(* CODESYS project geral_v2_1_0.library
   DefaultNamespace: Teknike_Geral
   DocFormat: reStructuredText
   Description: FBs de uso geral
   Author: Tiago B, Cunico
   Title: Geral
   Version: 2.1.0
   Company: Teknike
   Placeholder: Teknike_Geral

Project tree, tasks and I/O mapping:
  libraries: OSCAT - AixOCAT, * (RWTH Aachen University - E.ON Energy Research Center); Tc2_EtherCAT, * (Beckhoff Automation GmbH); Tc2_IoFunctions, * (Beckhoff Automation GmbH); Tc2_Standard, * (Beckhoff Automation GmbH); Tc2_System, * (Beckhoff Automation GmbH); Tc2_Utilities, * (Beckhoff Automation GmbH); Tc3_Database, * (Beckhoff Automation GmbH); Tc3_IPCDiag, * (Beckhoff Automation GmbH); Tc3_Module, * (Beckhoff Automation GmbH)
  DUTs/
    Ethercat/
      Cartoes/
      EtherCAT Diag/
        data type E_EcCommState
        data type ST_EcMasterDevState
        data type ST_PortAddr
        data type ST_SlaveState
        data type ST_SlaveStateInfo
        data type ST_SlaveStateInfoScanned
        data type ST_TopologyData
    data type st_Coluna
  FBs/
    Alarmes/
      GerenciadorSQL/
        data type EventosSQL
        function block FB_GerenciadorDeAlarmesSQL [ST]: FazTimeStamp, GeraTabela, GravaHistorico, LeHistorico
      GerenciadorV2/
        Duts/
          data type ST_Alarmes_Historico_V2
          data type ST_Alarmes_Online_V2
          data type ST_Alarmes_V2
        Mensagens/
          function block FB_MensagemMudouBool [ST]
          function block FB_MensagemMudouInt [ST]
          function block FB_MensagemMudouReal [ST]
        function block FB_GerenciadorAlarmesV2 [ST]: DesceAlarme, SobeAlarme
    Controle/
      BotaoDeParada/
        function block FB_BotaoParada [ST]
        data type st_BotaoParada
      Telerruptor/
        data type ConfigTelerruptor
        data type ConfigTelerruptorDB
        data type enum_GravaNomes
        data type enum_LeituradosNomes
        function block FB_IniciaOsBlocosDeConfigDoTelerruptor [ST]: GeraOsTelerruptores, GeraTabela, GravaValores, LeNomes
        function block FB_Telerruptor [ST]
        data type stTelerruptor
      function block FB_Cascata [ST]
      function block FB_Cascata1Ligado [ST]
      function block FB_ContaRPMporPulso [ST]
      function block FB_ControleTorreLuminosa [ST]
      function block FB_ControleTorreLuminosaV2 [ST]
      function block FB_TimerOnOff [ST]
      function block FB_TriggerDuplo [ST]
    CSV/
      data type eStatusCSV
      function block FB_ControleCSV [ST]: ExecutaEstado, TrocaEstado
      function block FB_EscreveCSV [ST]
      function block FB_EscreveCSVPonteiro [ST]
      function block FB_LeCSV [ST]
      data type st_ControleCSV
    Diagnostico/
      CAN/
        Sts/
          data type st_Diag_CAN
        function block fb_Diag_CAN [ST]
      Ethercat/
        function block FB_EtherCATDiag [ST]: M_CheckMasterDevState, M_GetScannedSlaveName_8, M_GetSlaveAdresses_1, M_GetSlaveIdentity_6, M_GetSlaveName_7, M_GetSlaveStates_2, M_GetTopoData_4, M_GetTopoDataLen_3, M_ScanSlaves_5
        function block FB_EtherCATFrameDiag [ST]
        data type st_DiagnosticoEthercat
      Ethernet_PCgeral/
        function block FB_Diag_Geral [ST]
        data type st_Diag_Ethernet
        data type st_Diag_PC_Geral
      KPI/
        function block FB_KPI_Geral [ST]
        data type st_KPI_Geral
    EAP/
      function block FB_HarmonizaVariavel_Bool [ST]
      function block FB_HarmonizaVariavel_Int [ST]
      function block FB_HarmonizaVariavel_Real [ST]
      function block FB_HeartBeat [ST]
    Emergencia/
      Sts/
        data type st_Emergencia
        data type st_Emergencia_Banco
        data type st_Emergencia_Config
        data type st_Emergencia_Entrada
        data type st_Emergencia_Saida
        data type st_TC_SAFE
      function block FB_Emergencia [ST]: AjeitaEntrada, AjeitaSaida, CalculaKPIs, FirstScan, Timers
    Geral/
      function block FB_FFT [ST]
      function block FB_HorimetroTime_Otimizado [ST]
      function block FB_HorimetroTime_Preciso [ST]
      function block FB_RodaTextoString [ST]
      function block FB_SalvaPersistentesEHoraAgora [ST]
    Graficos/
      GraficoTF2000/
        function block FB_GraficoTF2000 [ST]
        data type ST_Grafico
    Totalizador/
      Vazao/
        function block FB_TotalizadorVazao [ST]
        data type st_HistoricoHidrometro
    Valvulas/
      Proporcional/
        function block fb_ValvulaProporcional [ST]
        data type st_ValvulaProporcional
      Valvula/
        STs/
          data type st_EntradaValvula
          data type st_SaidaValvula
          data type st_Valvula
        function block FB_ControleValvula [ST]: Controle, Status
  FUNs/
    TempoParaString/
      function F_TempoEmStringAteHoras [ST]
    function F_ConcatArray [ST]
    function F_ConcatArray1000 [ST]
    function F_ConcatArray10000 [ST]
    function F_EntradaEmPorcentagem [ST]
    function F_EstruturaDiferente [ST]
    function F_LimpaArrayString [ST]
    function F_LimpaDataBase [ST]
    function F_MaisOuMenos [ST]
    function F_RetiraCasa [ST]
    function F_StringSeparadorArrayInt [ST]
    function F_StringSeparadorArrayInt_1 [ST]
  POUs/
    global variables GVL_BlibliotecaGeral
    program Main [ST]
    program ValidaLicensa [ST]: Licensas, Tempos
  Project Information/
    function F_GetCompany [ST]
    function F_GetTitle [ST]
    function F_GetVersion [ST]
  Version/
    global variables Global_Version
  VISUs/
*)

// DUTs/Ethercat/EtherCAT Diag/E_EcCommState
TYPE E_EcCommState : (
	eEcState_UNDEFINED 	:= 0,
	eEcState_INIT 		:= 1,
	eEcState_PREOP 		:= 2,
	eEcState_BOOT 		:= 3,
	eEcState_SAFEOP 	:= 4,
	eEcState_OP 		:= 8
);
END_TYPE

// DUTs/Ethercat/EtherCAT Diag/ST_EcMasterDevState
TYPE ST_EcMasterDevState :
STRUCT
	eEcState	 		: E_EcCommState;
	nReserved			: ARRAY [0..2] OF UINT;

	bLinkError			: BOOL;
	bResetRequired		: BOOL;
	bMissFrmRedMode		: BOOL;
	bWatchdogTriggerd	: BOOL;
	bDriverNotFound		: BOOL;
	bResetActive		: BOOL;
	bAtLeastOneNotInOp	: BOOL;
	bDcNotInSync		: BOOL;
END_STRUCT
END_TYPE

// DUTs/Ethercat/EtherCAT Diag/ST_PortAddr
TYPE ST_PortAddr :
STRUCT
	portA : UINT;
	portB : UINT;
	portC : UINT;
	portD : UINT;
END_STRUCT
END_TYPE

// DUTs/Ethercat/EtherCAT Diag/ST_SlaveState
TYPE ST_SlaveState :
STRUCT
	(* slave state *)
	eEcState 		: E_EcCommState;
	nReserved		: UINT;
	bError			: BOOL;
	bInvalidVPRS	: BOOL;
	nReserved2		: UINT;

	(* link state *)
	bNoCommToSlave	: BOOL;
	bLinkError		: BOOL;
	bMissingLink	: BOOL;
	bUnexpectedLink	: BOOL;
	bPortA			: BOOL;
	bPortB			: BOOL;
	bPortC			: BOOL;
	bPortD			: BOOL;
END_STRUCT
END_TYPE

// DUTs/Ethercat/EtherCAT Diag/ST_SlaveStateInfo
TYPE ST_SlaveStateInfo :
STRUCT
	nIndex 			: DINT;
	sName 			: STRING; 		(* name of slave given in System Manager *)
	sType 			: STRING;		(* type of slave, e.g. EK1100*)
	nECAddr 		: UINT;			(* EtherCAT Slave Addr *)
	bDiagData		: BOOL;			(* DiagData in Slave State *)
	stPortCRCErrors	: ST_EcCrcErrorEx;(* Slave CRC-Errors, separate for each Port *)
	nSumCRCErrors	: UDINT;		(* Slave CRC-Errors, sum of all Ports *)
	stState 		: ST_SlaveState;(* EtherCAT State and Link state*)
END_STRUCT
END_TYPE

// DUTs/Ethercat/EtherCAT Diag/ST_SlaveStateInfoScanned
TYPE ST_SlaveStateInfoScanned :
STRUCT
	nIndex 			: DINT;
	sName 			: STRING; 		(* name of slave given in System Manager *)
	sType 			: STRING;		(* type of slave, e.g. EK1100*)
	nECAddr 		: UINT;			(* EtherCAT Slave Addr *)
	bDifferentName	: BOOL;			(* Name of Scanned configuration differs from Configured configuration *)
	bDifferentType	: BOOL;			(* Type Of Scanned configuration differs from Configured configuration *)
	bDifferentAddr	: BOOL;			(* EcAddress of Scanned configuration differs from Configured configuration *)
END_STRUCT
END_TYPE

// DUTs/Ethercat/EtherCAT Diag/ST_TopologyData
TYPE ST_TopologyData :
STRUCT
	iOwnPhysicalAddr 	: UINT;
	iOwnAutoIncAddr		: UINT;
	stPhysicalAddr		: ST_PortAddr;
	stAutoIncAddr		: ST_PortAddr;
	iPortDelay			: ARRAY [0..2] OF UDINT; (* EC_AD, EC_DB, EC_BC *)
	iReserved			: ARRAY [0..7] OF UDINT;
END_STRUCT
END_TYPE

// DUTs/st_Coluna
TYPE st_Coluna :
STRUCT
	
	xComeca : BOOL;
	iOrdemCorLiga : ARRAY[1..6] OF INT; // array de qual corres ligam em qual ordem, 0 -> desligado 1 -> vermelho 2 -> amarelo 3 -> verde 4 -> azul 5 -> buzzer, se quiser que mais de um acione ao mesmo tempo so colocar os dois juntos tipo, verde e amarelo é 24 ou 42
	tTempoDeCadaAcionamento : ARRAY[1..6] OF TIME; // tempo que vai ser usado para cada item do iOrdemCorLiga
	

	xVermelho : BOOL;
	xAmarelo : BOOL;
	xAzul : BOOL;
	xVerde : BOOL;
	xBuzzer : BOOL;
	xErro : BOOL;
END_STRUCT
END_TYPE

// FBs/Alarmes/GerenciadorSQL/EventosSQL
TYPE EventosSQL :
STRUCT
	
	ID 				:	T_ULARGE_INTEGER;
	Data_On			:	STRING(80);	//Data de entrada do evento
	Hora_On			:	STRING(80);	//Hora de entrada do evento
	Data_Off		:	STRING(80);	//Data de saida do evento
	Hora_Off		:	STRING(80);	//Hora de saida do evento
	Tipo			:	INT;	//Hora de saida do evento
	TAG				:	STRING(80);	// tago do que deu problema
	Texto 			:	STRING(80);	// texto do alarme
	Usuario			:	STRING(80);	//UsuárioLogado
	Grupo			:	INT;			//Byte do grupo
	TimesTamp 		:	DT;



END_STRUCT
END_TYPE

// FBs/Alarmes/GerenciadorV2/Duts/ST_Alarmes_Historico_V2
TYPE ST_Alarmes_Historico_V2 : STRUCT

		sData_on  : STRING(20);  //Data de entrada do evento
		sData_off : STRING(20);  //Data de saida do evento
		sHora_on  : STRING(20);  //Hora de entrada do evento
		sHora_off : STRING(20);  //Hora de saida do evento
		iStatus   : INT;         //Byte do grupo
		sUsuario  : STRING;      //UsuárioLogado
		sTAG      : STRING;      //tag do que foi afetado
		sTexto    : STRING(255); //texto em si
		iTipo     : INT;         //mensagem ou alarme

	END_STRUCT
END_TYPE

// FBs/Alarmes/GerenciadorV2/Duts/ST_Alarmes_Online_V2
TYPE ST_Alarmes_Online_V2 : STRUCT

		sData          : STRING(20); //Hora de entrada do alarme
		sHora          : STRING(20); //Hora de saida do alarme
		sMensagem      : STRING(255); // mensagme que aparece na tela
		sUser          : STRING; // usuario
		iStatus        : INT; // se foi reconhecido como que ta
		iIdentificador : INT; // pra controle interno
		sTAG           : STRING; // tag do que foi afetado
		iTipo          : INT; // mensagem ou alarme

	END_STRUCT
END_TYPE

// FBs/Alarmes/GerenciadorV2/Duts/ST_Alarmes_V2
TYPE ST_Alarmes_V2 : STRUCT
		xAtivo : BOOL;
		sTexto : STRING(255);
		iTipo  : INT;
		sTAG   : STRING;
	END_STRUCT
END_TYPE

// FBs/Controle/BotaoDeParada/st_BotaoParada
TYPE st_BotaoParada :
STRUCT
	xSinalBP_IN		: BOOL;
	xSinalBP_OUT	: BOOL;
	xLedBP			: BOOL;
END_STRUCT
END_TYPE

// FBs/Controle/Telerruptor/ConfigTelerruptor
TYPE ConfigTelerruptor :
STRUCT RETAIN PERSISTENT
		sNome_Funcao				: STRING;
		rTempoTelerruptorAcionado 	: REAL;
END_STRUCT
END_TYPE

// FBs/Controle/Telerruptor/ConfigTelerruptorDB
TYPE ConfigTelerruptorDB :
STRUCT
	Telerruptor: DINT;
	Tag: STRING(80);
	Funcao: STRING(80);
END_STRUCT
END_TYPE

// FBs/Controle/Telerruptor/enum_GravaNomes
{attribute 'qualified_only'}
{attribute 'strict'}
TYPE enum_GravaNomes :
(
	eEsperando := 0,
	eAbreConexao := 1,
	eGravaNomes := 2,
	eCriaComando := 3,
	eFechaConexao := 4,
	eParado := 100
);
END_TYPE

// FBs/Controle/Telerruptor/enum_LeituradosNomes
{attribute 'qualified_only'}
{attribute 'strict'}
TYPE enum_LeituradosNomes :
(
	eEsperando := 0,
	eAbreConexao := 1,
	eLeOsNomes := 2,
	eMonitoraTrocaDeNomes := 3,
	eFechaConexao := 4,
	eParado := 100
);
END_TYPE

// FBs/Controle/Telerruptor/stTelerruptor
TYPE stTelerruptor :
STRUCT
	xFeedBackTelerruptor 		: BOOL;
	xLigaIHM		 			: BOOL;
	xLigaBotoeira				: BOOL;
	xLigaInterruptor			: BOOL;
	xAcionaTelerruptor			: BOOL;
	Config						: ConfigTelerruptor;
END_STRUCT
END_TYPE

// FBs/CSV/eStatusCSV
//{attribute 'qualified_only'}
{attribute 'strict'}
TYPE eStatusCSV :
(
	Esperando := 0,
	ChecandoCaminhoGeral,
	ChecandoCaminhoEspecifico,
	Gravando,
	lendoArquivos,
	Lendo,
	Erro
);
END_TYPE

// FBs/CSV/st_ControleCSV
TYPE st_ControleCSV :
STRUCT
	
	xLeCSV 						: BOOL;
	xEscreveCSV 				: BOOL;
	xEscolhidoArquivo			: BOOL;
	
	sArquivosSelecionado		: STRING(255);

	xEscritaOcupado 			: BOOL;
	xLeituraOcupado 			: BOOL;
	
	
	iTotalLeitura 				: INT;
	iAtualLeitura 				: INT;
	iTotalEscrita 				: INT;
	iAtualEscrita 				: INT;
	sArquivos					: ARRAY[1..20]  OF STRING(255);
	
	sStado : eStatusCSV;

END_STRUCT
END_TYPE

// FBs/Diagnostico/CAN/Sts/st_Diag_CAN
TYPE st_Diag_CAN :
	STRUCT
		//Linkar no device
		usError				AT %I*	: USINT;	// numero de Box com erro
		uCanState			AT %I*	: UINT;		// gera outros bits
		usRxErrorCounter	AT %I*	: USINT;	// contagem 
		usTxErrorCounter	AT %I*	: USINT;	// contagem
		diagFlag			AT %I*	: BIT;

		//Linkar nos nos
		uNodeState AT %I* : ARRAY[1..126] OF USINT;

		//Gerado apartir do CAN state
		xBusOFF			: BOOL;
		xCanWarning		: BOOL;
		xRxOverrun		: BOOL;
		xCANSendError	: BOOL;
		xFilaRxOverflow	: BOOL;
		xFilaTxOverflow	: BOOL;

		xNoOk		: ARRAY[1..126] OF BOOL;
		sEstadoNo	: ARRAY[1..126] OF STRING;

	END_STRUCT
END_TYPE

// FBs/Diagnostico/Ethercat/st_DiagnosticoEthercat
TYPE st_DiagnosticoEthercat :
	STRUCT

		(* ******************* EtherCAT Frame ***************************** *)
		fbEtherCATFrameDiag	: FB_EtherCATFrameDiag;	// frame diagnostic 
		wFrmXWcState AT %I*	: WORD;					// link to task related ethercat frame state (Frm1WcState)
		wReqZeroMask		: WORD := 16#FFFF;		// clear bit to ignore datagram error of Frm1WcState
		bFrameWcStateOK		: BOOL;					// this frame is OK 

		(* ******************* EtherCAT Diag ***************************** *)
		bEtherCATOK				: BOOL;					// no problem on EtherCAT
		bFrameWcStateError		: BOOL;					// at least one fram with error
		bSlaveCountError		: BOOL;					// EtherCAT slave count mismatch (# of cfg slaves <> # of found slaves)
		bMasterDevStateError	: BOOL;					// EtherCAT master device state signals error
		bBarramentoInterrompido	: BOOL;					// caso o barramento esteja interrompido
		stMasterDevState		: ST_EcMasterDevState;	// device state split to a structure
		bBusy					: BOOL;					// diagnostic FB is busy
		bError					: BOOL;					// diagnostic FB has an error
		iErrorID				: UDINT;				// error ID of diagnostic FB

		(* cyclic variables from EtherCAT Master *)
		nEcMasterSlaveCount		AT %I*	: UINT;				// link to SlaveCount of EtherCAT Master (Inputs)
		nEcMasterSlaveCount2	AT %I*	: UINT;				// link to SlaveCount of EtherCAT Master (Inputs)
		nEcMasterDevState		AT %I*	: UINT;				// link to DevState of EtherCAT Master (Inputs)
		nEcMasterDeviceId		AT %I*	: UINT;				// link to DevID of EtherCAT Master (InfoData)
		arrEcMasterNetId		AT %I*	: T_AmsNetIdArr;	// link to NetID of EtherCAT Master (InfoData)
		sEcMasterNetId					: T_AmsNetId := '';
		nEcMasterSlaveCountCfg AT %I*	: UINT; // link to CfgSlaveCount of EtherCAT Master (InfoData)

		(* general variables *)
		arrDiagSlaveInfo		: ARRAY[0..255] OF ST_SlaveStateInfo;			// read in info of configured EtherCAT slaves 
		arrDiagSlaveInfoScanned	: ARRAY[0..255] OF ST_SlaveStateInfoScanned;	// read in info of scanned EtherCAT slaves

	END_STRUCT
END_TYPE

// FBs/Diagnostico/Ethernet_PCgeral/st_Diag_Ethernet
TYPE st_Diag_Ethernet :
STRUCT
	
	sNome 			: STRING;
	sNomeAdaptador 	: STRING;
	sIP				: STRING;
	sMask 			: STRING;
	xDHCP 			: BOOL;

END_STRUCT
END_TYPE

// FBs/Diagnostico/Ethernet_PCgeral/st_Diag_PC_Geral
TYPE st_Diag_PC_Geral :
STRUCT
	
	//Rede
	NumeroDePortasRede	: USINT;
	stEthernet : ARRAY[1..20] OF st_Diag_Ethernet;
	
	//CPU
	uiUsoCpu : UINT;
	iTempCpu : INT;
	rMemoriaRamUsada : REAL;
	rEspacoLivreHD : REAL;
	sNomeCPU : STRING;
	
	//Twincat
	tcVersion : STRING;
	tcAMSNetID : STRING;
	tcSystemID : STRING;
	


END_STRUCT
END_TYPE

// FBs/Diagnostico/KPI/st_KPI_Geral
TYPE st_KPI_Geral :
	STRUCT
		stGraficoIHM : ARRAY[0..2] OF ST_Grafico;
	
		rPorcEstado1	: REAL;
		rPorcEstado2	: REAL;
		rPorcEstado3	: REAL;

		tEstado1	: TIME;
		tEstado2	: TIME;
		tEstado3	: TIME;
	END_STRUCT
END_TYPE

// FBs/Emergencia/Sts/st_Emergencia
TYPE st_Emergencia :
STRUCT
	En : st_Emergencia_Entrada;
	Sa : st_Emergencia_Saida;
	Config : st_Emergencia_Config;
	Banco : st_Emergencia_Banco;
	Safe : st_TC_SAFE;
END_STRUCT
END_TYPE

// FBs/Emergencia/Sts/st_Emergencia_Banco
TYPE st_Emergencia_Banco :
STRUCT
		Emergencia	: T_ULARGE_INTEGER;
		Tag			: STRING(80);
		Funcao		: STRING(80);
		Timestamp	: DT;
END_STRUCT
END_TYPE

// FBs/Emergencia/Sts/st_Emergencia_Config
TYPE st_Emergencia_Config :
STRUCT RETAIN PERSISTENT
	xControleInterno : BOOL;
	xbypassCH2 : BOOL;
	tDiscrepancia : TIME;
	xControleTCSafe : BOOL;
END_STRUCT
END_TYPE

// FBs/Emergencia/Sts/st_Emergencia_Entrada
TYPE st_Emergencia_Entrada :
STRUCT
	xCH1 : BOOL;
	xCH2 : BOOL;
	xEmergenciaOK : BOOL; // status da emergencia, se for externa tb serve
	sNomeFuncao : STRING;
	xReset : BOOL;
	xResetFisico : BOOL;
	stHoraAgora : TIMESTRUCT;
END_STRUCT
END_TYPE

// FBs/Emergencia/Sts/st_Emergencia_Saida
TYPE st_Emergencia_Saida :
STRUCT	
	kpi : ARRAY[0..23] OF st_KPI_Geral;
	xErro : BOOL;
	xLedReset : BOOL;
	sEstadoIHM : STRING;
	iStatus : INT;//0 : desligado, 1 : OK, 2 : Esperando Reset, 3 : Desincronizado, 4 : EDM, 5 : Outro Erro
END_STRUCT
END_TYPE

// FBs/Emergencia/Sts/st_TC_SAFE
TYPE st_TC_SAFE :
STRUCT
	RESET 		AT%Q* 	: BOOL;
	EDM 		AT%Q*	: BOOL;
	RUN			AT%Q*	: BOOL;
	ERRACK		AT%Q*	: BOOL;
	
	State		AT%I*	: USINT;
	Diag		AT%I*	: UINT;
END_STRUCT
END_TYPE

// FBs/Graficos/GraficoTF2000/ST_Grafico
TYPE ST_Grafico :
STRUCT
	x : STRING;
	y : REAL;
	label : STRING(255);
	sCor : STRING(255);//Cor em Hexa
	sTipo: STRING;//sendo eles "line", "bar", "scatter", "bubble", "pie", "doughnut", "polarArea" 
END_STRUCT
END_TYPE

// FBs/Totalizador/Vazao/st_HistoricoHidrometro
TYPE st_HistoricoHidrometro :
STRUCT
	sDataHora : STRING;
	rTotal : REAL;
	rDiferenca : REAL;
END_STRUCT
END_TYPE

// FBs/Valvulas/Proporcional/st_ValvulaProporcional
TYPE st_ValvulaProporcional :
STRUCT RETAIN PERSISTENT
	xManu : BOOL;
	rValorManu : REAL;
	rValorAuto : REAL;
	
	rMinimo : REAL := 0;
	rMaximo : REAL := 32767;
	rValorDeSaida : REAL;
	
	
	rPorcentSaida : REAL;
	
	iStsValvula  : INT;
	
	sNomeFuncao : STRING;
	
	
END_STRUCT
END_TYPE

// FBs/Valvulas/Valvula/STs/st_EntradaValvula
TYPE st_EntradaValvula :
STRUCT
	xAutomaticoManual 	: BOOL;
	xLigaManu			: BOOL;
	xLigaAuto			: BOOL;
	xBloqueio			: BOOL;
	xEmergenciaOK		: BOOL;
	xFeedBackValvula	: BOOL;
	xByPassFeedBack		: BOOL;
	xResetContador		: BOOL;
	rTempoFeedBackSeg	: REAL;
	sNome_Funcao		: STRING;
	xNormalmenteAberto	: BOOL;
	i					: INT;
END_STRUCT
END_TYPE

// FBs/Valvulas/Valvula/STs/st_SaidaValvula
TYPE st_SaidaValvula :
STRUCT
	xSaidaValvula		: BOOL;
	iStsValvula			: INT;
	iSucessoAionamento	: INT;
	iFalhaAcionamento	: INT;
END_STRUCT
END_TYPE

// FBs/Valvulas/Valvula/STs/st_Valvula
TYPE st_Valvula :
STRUCT
	en : st_EntradaValvula;
	sa : st_SaidaValvula;
END_STRUCT
END_TYPE

// POUs/GVL_BlibliotecaGeral
//{attribute 'qualified_only'}
VAR_GLOBAL
	
    {attribute 'hide'} 
	{attribute 'tc_no_symbol'}
	xLicensaValida87208720 : BOOL;
	LicensaValida : BOOL;
	STCheckLicense : ST_CheckLicense;
END_VAR

// Version/Global_Version
{attribute 'TcGenerated'}
{attribute 'no-analysis'}
{attribute 'linkalways'}
// This function has been automatically generated from the project information.
VAR_GLOBAL CONSTANT
	{attribute 'const_non_replaced'}
	stLibVersion_Geral : ST_LibVersion := (iMajor := 2, iMinor := 1, iBuild := 0, iRevision := 0, nFlags := 0, sVersion := '2.1.0');
END_VAR

// FBs/Alarmes/GerenciadorSQL/FB_GerenciadorDeAlarmesSQL
//{attribute 'hide_all_locals'}
FUNCTION_BLOCK FB_GerenciadorDeAlarmesSQL
VAR_IN_OUT
	arrayAlarmes	: ARRAY[*] OF ST_Alarmes_V2;
	Alarmes_Online	: ARRAY[*] OF ST_Alarmes_Online_v2;
	HistoricoSQL	: ARRAY[*] OF EventosSQL;
	RT				: ARRAY[*] OF R_TRIG;	//
	FT				: ARRAY[*] OF F_TRIG;	//
END_VAR
VAR_INPUT
	xReconhece		: BOOL;
	sUsuario		: STRING;
	sNomeTabela		: STRING;
	iNumeroDataBase	: INT := 1;
	xCriaTabela		: BOOL;
	stTempoAgora	: TIMESTRUCT;
END_VAR
VAR_OUTPUT
	xAlarmeAtivo			: BOOL;
	xAlarmeAtivoReconhecido	: BOOL;
	sErro					: STRING;
END_VAR
VAR
	VariavelParaTamanhoNoBloco : EventosSQL;

	// Erros
	xAbaixoOk		: BOOL	:= TRUE;
	xAcimaOK		: BOOL	:= TRUE;
	xHistoricoOk	: BOOL	:= TRUE;

	// variaveis para controle dos loops
	iMaxAlarmesOnline		: INT;
	iMaxAlarmesHistorico	: INT;

	//Ler dados da tabela usando o bloco Read Struct
	fbPLCDBRead		: FB_PLCDBReadEvt(sNetID := '', tTimeout := T#30S);	//Bloco para leitura do banco de dados sem filtro
	sMensagemErro1	: STRING;											//Mensagem de erro

	ColumnNames : ARRAY[0..10] OF STRING(50) := ['ID',
												'Data_On',
												'Hora_On',
												'Data_Off',
												'Hora_Off',
												'Tipo',
												'TAG',
												'Texto',
												'Usuario',
												'Grupo',
												'Timestamp'];

	xEscreve	: BOOL;
	xAtualiza	: BOOL;

	// fb do gerenciador e auxiliares
	GerenciaAlarmes : FB_GerenciadorAlarmesV2;
	//para a data e hora
	sData	: ARRAY[1..5] OF STRING(255);
	sHora	: ARRAY[1..7] OF STRING(255);

	// para controle do historico e da escrita dele no SQL
	Alarmes_Historico		: ARRAY[0..1000] OF ST_Alarmes_Historico_v2;	// esse é o atual
	Alarmes_Historico_Bufer	: ARRAY[0..1000] OF ST_Alarmes_Historico_v2;	// Buffer pra escrita quando varios alarmes caiem de uma vez so
	Alarmes_Historico_Aux	: ARRAY[0..1000] OF ST_Alarmes_Historico_v2;	// esse é pra ver see é diferente
	tofEsperaAlarme			: TOn;

	//Gravar dados na tabela
	fbPLCDBWrite			: FB_PLCDBWriteEvt(sNetID := '', tTimeout := T#30S);	//Bloco para gravar no banco de dados
	systime					: GETSYSTEMTIME;										//Faz a leitura da data e hora do sistema
	currentTime				: T_FILETIME;
	bGravarDados			: BOOL;
	sMensagemErroEscrita	: STRING;
	AuxEscreve				: EventosSQL;
	coutBuffer				: INT;
	rtComecaEscever			: R_TRIG;
	ftTerminouDeGravar		: F_TRIG;
	xAtualizado				: BOOL;
	xTemQueEscrever			: BOOL;
	iDeslocamenteAjuste		: INT;

	// geral
	i				: INT;
	xPrimeiroScan	: BOOL := TRUE;

	rtCria			: R_TRIG;
	xCria			: BOOL;
	fbPLCDBCreate	: FB_PLCDBCreateEvt(sNetID := '', tTimeout := T#30S);

	ColumnInfo : ARRAY[0..10] OF ST_ColumnInfo := [(sName := 'ID', eType := E_ColumnType.BigInt, nLength := 8, sProperty := 'IDENTITY(1,1)'),
													(sName := 'Data_On', eType := E_ColumnType.NVarChar, nLength := 80),
													(sName := 'Hora_On', eType := E_ColumnType.NVarChar, nLength := 80),
													(sName := 'Data_Off', eType := E_ColumnType.NVarChar, nLength := 80),
													(sName := 'Hora_Off', eType := E_ColumnType.NVarChar, nLength := 80),
													(sName := 'Tipo', eType := E_ColumnType.SmallInt, nLength := 2),
													(sName := 'TAG', eType := E_ColumnType.NVarChar, nLength := 80),
													(sName := 'Texto', eType := E_ColumnType.NVarChar, nLength := 80),
													(sName := 'Usuario', eType := E_ColumnType.NVarChar, nLength := 80),
													(sName := 'Grupo', eType := E_ColumnType.SmallInt, nLength := 2),
													(
				sName := 'Timestamp',
					eType := E_ColumnType.DateTime,
					nLength := 4,
					sProperty := 'DEFAULT CURRENT_TIMESTAMP ON UPDATE CURRENT_TIMESTAMP')];
					
	tonPodeLer : TON;

END_VAR


IF xLicensaValida87208720 THEN
	

	// ve se os tamanhos dos arrays estao ok
	xAbaixoOk		:= LOWER_BOUND(arrayAlarmes, 1) = 0 AND LOWER_BOUND(arrayAlarmes, 1) = LOWER_BOUND(Alarmes_Online, 1);
	xAcimaOK		:= UPPER_BOUND(arrayAlarmes, 1) = UPPER_BOUND(Alarmes_Online, 1);
	xHistoricoOk	:= LOWER_BOUND(HistoricoSQL, 1) = 0;
	
	GeraTabela();
	
	IF xAbaixoOk AND xAcimaOK AND xHistoricoOk THEN
	
		IF xPrimeiroScan THEN
			FazTimeStamp();
			systime(timeLoDw => currentTime.dwLowDateTime, timeHiDW => currentTime.dwHighDateTime);
			// troca a variavel pra ficar bom pro sql
			AuxEscreve.Data_Off		:= '';
			AuxEscreve.Data_On		:= F_ConcatArray(sData);
			AuxEscreve.Hora_Off		:= '';
			AuxEscreve.Hora_On		:= F_ConcatArray(sHora);
			AuxEscreve.Usuario		:= '';
			AuxEscreve.Texto		:= 'CPU ligou';
			//AuxEscreve.TimesTamp	:= FILETIME_TO_DT(currentTime) - (T#3H);
	
			xAtualiza	:= TRUE;
			xEscreve	:= TRUE;
	
			iMaxAlarmesOnline		:= TO_INT(UPPER_BOUND(Alarmes_Online, 1));
			iMaxAlarmesHistorico	:= TO_INT(UPPER_BOUND(HistoricoSQL, 1));
		END_IF
	
		LeHistorico();
		FazTimeStamp();
		GravaHistorico();
	
		GerenciaAlarmes
			(
				Alarmes_Array := arrayAlarmes,
					Alarmes_Online := Alarmes_Online,
					Alarmes_Historico := Alarmes_Historico,
					RT := RT,
					FT := FT,
					xReconheceAlarmes := xReconhece,
					sData := F_ConcatArray(sData),
					sHora := F_ConcatArray(sHora),
					sUser := sUsuario,
					xAlarmeAtivo => xAlarmeAtivo,
					xAlarmeAtivoReconhecido => xAlarmeAtivoReconhecido);
	
		// independente se tem so um diferente ou varios, esse if sempre sera verdade
		IF Alarmes_Historico[0].sHora_off <> Alarmes_Historico_Aux[0].sHora_off AND NOT (Alarmes_Historico[0].sHora_off = '') THEN
			FOR i := 0 TO 1000 DO
				// quando nao tiver alguma coisa na posição do buffer ele sai do for
				IF (Alarmes_Historico_Bufer[i].sHora_off = '') THEN
					EXIT;
				END_IF
			END_FOR
			// e joga aqui o valor de i que é a primeira posição que nao tem na da no buffer
			coutBuffer := i;
			// deslocamente para ajustar o index conforme vai passando e encontrando alarmes diferentes
			iDeslocamenteAjuste := 0;
	
			// passa por todo os alarmes vendo quem ta acionado e joga no buffer
			FOR i := 0 TO 1000 DO
				IF Alarmes_Historico[i].sHora_off <> Alarmes_Historico_Aux[i - iDeslocamenteAjuste].sHora_off
						AND NOT (Alarmes_Historico[i].sHora_off = '') THEN
					Alarmes_Historico_Bufer[coutBuffer]	:= Alarmes_Historico[i];
					coutBuffer							:= coutBuffer + 1;
					iDeslocamenteAjuste					:= iDeslocamenteAjuste + 1;
				ELSE
					//IF THEN
	
					//ELSE
					EXIT;
					//END_IF
				END_IF
			END_FOR
		END_IF
	
		Alarmes_Historico_Aux := Alarmes_Historico; // atualiza para o atual
	
		// da o start quando chega o primeiro item pra ler no buffer
		rtComecaEscever(CLK := (Alarmes_Historico_Bufer[0].sHora_off <> ''), Q =>);
	
		IF rtComecaEscever.q THEN
			xEscreve	:= TRUE;
			xAtualizado	:= FALSE;
	
			// faz esse esquema a primeira vez
			// pega o tempo de agora
			systime(timeLoDw => currentTime.dwLowDateTime, timeHiDW => currentTime.dwHighDateTime);
			// troca a variavel pra ficar bom pro sql
			AuxEscreve.Data_Off	:= Alarmes_Historico_Bufer[0].sData_off;
			AuxEscreve.Data_On	:= Alarmes_Historico_Bufer[0].sData_On;
			AuxEscreve.Hora_Off	:= Alarmes_Historico_Bufer[0].sHora_Off;
			AuxEscreve.Hora_On	:= Alarmes_Historico_Bufer[0].sHora_On;
			AuxEscreve.Usuario	:= Alarmes_Historico_Bufer[0].sUsuario;
			AuxEscreve.TAG		:= Alarmes_Historico_Bufer[0].sTAG;
			AuxEscreve.Texto	:= Alarmes_Historico_Bufer[0].sTexto;
			AuxEscreve.Grupo	:= Alarmes_Historico_Bufer[0].iStatus;
			AuxEscreve.Tipo		:= Alarmes_Historico_Bufer[0].iTipo;
	
		END_IF
	
		ftTerminouDeGravar(CLK := xEscreve, Q =>);
	
		IF ftTerminouDeGravar.q THEN
			FOR i := 0 TO 999 DO
				Alarmes_Historico_Bufer[i] := Alarmes_Historico_Bufer[i + 1];
	
				IF Alarmes_Historico_Bufer[i].sHora_off = '' THEN
					EXIT;
				END_IF
			END_FOR
	
			xAtualizado := TRUE;
		END_IF
	
		IF NOT xEscreve AND xAtualizado AND Alarmes_Historico_Bufer[0].sHora_off <> '' THEN
	
			// pega o tempo de agora
			systime(timeLoDw => currentTime.dwLowDateTime, timeHiDW => currentTime.dwHighDateTime);
			// troca a variavel pra ficar bom pro sql
			AuxEscreve.Data_Off	:= Alarmes_Historico_Bufer[0].sData_off;
			AuxEscreve.Data_On	:= Alarmes_Historico_Bufer[0].sData_On;
			AuxEscreve.Hora_Off	:= Alarmes_Historico_Bufer[0].sHora_Off;
			AuxEscreve.Hora_On	:= Alarmes_Historico_Bufer[0].sHora_On;
			AuxEscreve.Usuario	:= Alarmes_Historico_Bufer[0].sUsuario;
			AuxEscreve.TAG		:= Alarmes_Historico_Bufer[0].sTAG;
			AuxEscreve.Texto	:= Alarmes_Historico_Bufer[0].sTexto;
			AuxEscreve.Grupo	:= Alarmes_Historico_Bufer[0].iStatus;
	
			//manda escrever
			xEscreve := TRUE;
			// tira esse bit pra esperar atualizar
			xAtualizado := FALSE;
		END_IF
	
		tofEsperaAlarme.in := TRUE;
	
		IF tofEsperaAlarme.q THEN
			xAtualiza			:= TRUE;
			tofEsperaAlarme.in	:= FALSE;
		END_IF
	
		tofEsperaAlarme(IN :=, PT := T#1S, Q =>, ET =>);
	
		xPrimeiroScan := FALSE;
	
	ELSE
		sErro := '';
	
		IF xHistoricoOk THEN
			sErro := 'historico precisa começar em 0';
		END_IF
	
		IF xAbaixoOk THEN
			sErro := 'tanto o online quanto o alarmes precisa começar em 0';
		END_IF
	
		IF xAcimaOK THEN
			sErro := 'tanto o online quanto o alarmes ter o mesmo tamanho';
		END_IF
	
	END_IF
	
ELSE
	ValidaLicensa();
END_IF

ACTION FazTimeStamp:



IF xPrimeiroScan THEN
	systime(timeLoDw => currentTime.dwLowDateTime, timeHiDW => currentTime.dwHighDateTime);
	AuxEscreve.TimesTamp := (FILETIME_TO_DT(currentTime));
	stTempoAgora := DT_TO_SYSTEMTIME(FILETIME_TO_DT(currentTime) - (T#3h));
END_IF

systime(timeLoDw => currentTime.dwLowDateTime, timeHiDW => currentTime.dwHighDateTime);
AuxEscreve.TimesTamp := (FILETIME_TO_DT(currentTime));


IF stTempoAgora.wDay < 10 THEN
	sData[1] := concat('0', TO_STRING(stTempoAgora.wDay));
ELSE
	sData[1] := WORD_TO_STRING(stTempoAgora.wDay);
END_IF

sData[2] := '/';

IF stTempoAgora.wMonth < 10 THEN
	sData[3] := concat('0', TO_STRING(stTempoAgora.wMonth));
ELSE
	sData[3] := WORD_TO_STRING(stTempoAgora.wMonth);
END_IF

sData[4] := '/';

sData[5] := TO_STRING(stTempoAgora.wYear);

IF stTempoAgora.wHour < 10 THEN
	sHora[1] := concat('0', TO_STRING(stTempoAgora.wHour));
ELSE
	sHora[1] := WORD_TO_STRING(stTempoAgora.wHour);
END_IF

sHora[2] := ':';

IF stTempoAgora.wMinute < 10 THEN
	sHora[3] := concat('0', TO_STRING(stTempoAgora.wMinute));
ELSE
	sHora[3] := WORD_TO_STRING(stTempoAgora.wMinute);
END_IF

sHora[4] := ':';

IF stTempoAgora.wSecond < 10 THEN
	sHora[5] := concat('0', TO_STRING(stTempoAgora.wSecond));
ELSE
	sHora[5] := WORD_TO_STRING(stTempoAgora.wSecond);
END_IF

sHora[6] := '.';

IF stTempoAgora.wMilliseconds < 100 THEN
	IF stTempoAgora.wMilliseconds < 10 THEN
		sHora[7] := concat('00', TO_STRING(stTempoAgora.wMilliseconds));
	ELSE
		sHora[7] := concat('0', TO_STRING(stTempoAgora.wMilliseconds));
	END_IF
ELSE
	sHora[7] := WORD_TO_STRING(stTempoAgora.wMilliseconds);
END_IF
END_ACTION

ACTION GeraTabela:

rtCria(CLK := xCriaTabela, Q =>);

IF rtCria.q THEN
	xCria := TRUE;
END_IF

IF xCria THEN

	IF fbPLCDBCreate.Table(
			hDBID := INT_TO_UDINT(iNumeroDataBase),
			sTableName := sNomeTabela,
			pTableCfg := ADR(ColumnInfo),
			cbTableCfg := SIZEOF(ColumnInfo))
	THEN
		xCria := FALSE;
	END_IF

END_IF
END_ACTION

ACTION GravaHistorico:

IF xEscreve THEN
	IF fbPLCDBWrite.WriteStruct(
			hDBID := int_to_Udint(iNumeroDataBase),
			sTableName := sNomeTabela,
			pRecord := ADR(AuxEscreve),
			cbRecord := SIZEOF(AuxEscreve),
			pColumnNames := ADR(ColumnNames),
			cbColumnNames := SIZEOF(ColumnNames))
	THEN
		IF fbPLCDBWrite.bError THEN
			sMensagemErroEscrita := 'Erro ao gravar no banco de dados';
			xEscreve             := FALSE;
		ELSE
			sMensagemErroEscrita := 'Dados gravados com sucesso';
			xEscreve             := FALSE;
		END_IF
	END_IF
END_IF
END_ACTION

ACTION LeHistorico:

tonPodeLer(IN:= NOT xEscreve, PT:= T#1S, Q=> , ET=> );

IF xAtualiza AND tonPodeLer.q THEN
	IF fbPLCDBRead.ReadStruct(
			hDBID := INT_TO_UDINT(iNumeroDataBase),
			sTableName := sNomeTabela,
			pColumnNames := ADR(ColumnNames),
			cbColumnNames := SIZEOF(ColumnNames),
			sOrderByColumn := ColumnNames[0],
			eOrderType := E_OrderType.DESC,
			nStartIndex := 0,
			nRecordCount := INT_TO_UDINT(iMaxAlarmesHistorico),
			pData := (HistoricoSQL),
			cbData := SIZEOF(VariavelParaTamanhoNoBloco) * 1000)
	THEN

		IF fbPLCDBRead.bError THEN
			sMensagemErro1 := 'Erro ao ler o banco de dados';
			xAtualiza      := FALSE;
		ELSE
			sMensagemErro1 := 'Leitura dos dados com sucesso';
			xAtualiza      := FALSE;
		END_IF
	END_IF

END_IF
END_ACTION

END_FUNCTION_BLOCK

// FUNs/F_ConcatArray
FUNCTION F_ConcatArray : string(255) //Concatena um array de string
VAR_IN_OUT
	sArray : ARRAY[*] OF STRING(255);
END_VAR
VAR
	iTamanhoArray : INT;
	iTamanhoMinArray : INT;
	i : INT;
END_VAR



IF xLicensaValida87208720 THEN	
	
	
	//Criado por Tiago Bortolini Cunico
	
	iTamanhoArray := DINT_TO_INT(UPPER_BOUND(sArray,1));
	iTamanhoMinArray := DINT_TO_INT(LOWER_BOUND(sArray,1));
	
	FOR i := iTamanhoMinArray TO iTamanhoArray DO
		F_ConcatArray := CONCAT(F_ConcatArray,sArray[i]);
	END_FOR

ELSE
	F_ConcatArray := '';
	ValidaLicensa();
END_IF

END_FUNCTION

// POUs/ValidaLicensa
PROGRAM ValidaLicensa
VAR
	
fb1 : FB_GerenciadorDeAlarmesSQL;
Tempo : FB_HorimetroTime_Otimizado;
geral : FB_SalvaPersistentesEHoraAgora;
fbCoraca : FB_HeartBeat;
fbxHarmoniza : FB_HarmonizaVariavel_Bool;
fbiHarmoniza : FB_HarmonizaVariavel_int;
fbrHarmoniza : FB_HarmonizaVariavel_real;
fbKPI : FB_KPI_Geral;
fbEmergencia : FB_Emergencia;

{attribute 'tc_no_symbol'}
Olhaliscensa : FB_CheckLicense;
{attribute 'tc_no_symbol'}
GUIDLicensa : GUID := STRING_TO_GUID('86E801DA-D766-479A-B8BD-B88BF7CB0709');


END_VAR




Licensas();

STCheckLicense := Olhaliscensa.stCheckLicense;

xLicensaValida87208720 :=
 Olhaliscensa.stCheckLicense.eResult = 0 OR// essa é so pros que sao da beckhoff mesmo
 Olhaliscensa.stCheckLicense.eResult = 16#203 OR
 Olhaliscensa.stCheckLicense.eResult = 16#254 OR
 Olhaliscensa.stCheckLicense.eResult = 16#255;

 LicensaValida := xLicensaValida87208720;

ACTION Licensas:
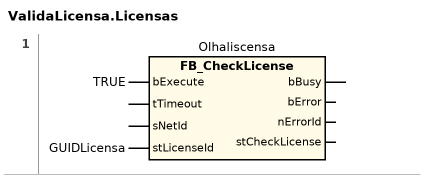
// NETWORK 1
Olhaliscensa(bExecute := TRUE, stLicenseId := GUIDLicensa); // FB_CheckLicense
END_ACTION

ACTION Tempos:
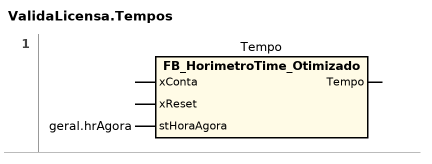
// NETWORK 1
Tempo(stHoraAgora := geral.hrAgora); // FB_HorimetroTime_Otimizado
END_ACTION

END_PROGRAM

// FBs/Geral/FB_HorimetroTime_Otimizado
FUNCTION_BLOCK FB_HorimetroTime_Otimizado
VAR_INPUT
	xConta : BOOL;
	xReset : BOOL;
	stHoraAgora : TIMESTRUCT;
END_VAR
VAR_OUTPUT
	Tempo : TIME;
END_VAR
VAR

	rtReset : R_TRIG;
	
	stHoraAnterior : TIMESTRUCT;


END_VAR


IF xLicensaValida87208720 THEN

	
	rtReset(CLK:= xReset, Q=> );
	
	IF rtReset.q THEN
		Tempo := T#0S;
	END_IF
	
	
	IF (stHoraAgora.wSecond <> stHoraAnterior.wSecond) AND xConta THEN
		Tempo := Tempo + T#1S;
	END_IF
	
	stHoraAnterior := stHoraAgora;

ELSE
	ValidaLicensa();
END_IF

END_FUNCTION_BLOCK

// FBs/Geral/FB_SalvaPersistentesEHoraAgora
FUNCTION_BLOCK FB_SalvaPersistentesEHoraAgora
VAR_INPUT
END_VAR
VAR_OUTPUT
	hrAgora : TIMESTRUCT;
END_VAR
VAR	
	EscrevePersistente : FB_WritePersistentData;
	fbLocalSystemTime: FB_LocalSystemTime;
END_VAR


IF xLicensaValida87208720 THEN
		
	
	
	fbLocalSystemTime(
		sNetID:= , 
		bEnable:= TRUE, 
		dwCycle:= , 
		dwOpt:= , 
		tTimeout:= T#5S, 
		bValid=> , 
		systemTime=> hrAgora, 
		tzID=> );
	
	
	EscrevePersistente(
		NETID:= , 
		PORT:= 851, 
		START:= hrAgora.wMinute MOD 5 = 0, 
		TMOUT:= , 
		MODE:= , 
		BUSY=> , 
		ERR=> , 
		ERRID=> );


ELSE
	ValidaLicensa();
END_IF

END_FUNCTION_BLOCK

// FBs/EAP/FB_HeartBeat
FUNCTION_BLOCK FB_HeartBeat
VAR_INPUT
	xHeartBeatEntrada 	: BOOL; // HeartBeat que precisa ser monitorado
	xTK2000				: BOOL; //bool para controle da saida das imagens
	tTempoAlive 		: TIME := T#50MS; // Definição tempo ate ser considerado morto (Por padrão é 50ms )
	uiQualidade			: UINT;	// variavel que mostra a qualidade das variaveis, se for > 0 é pq ja deu ruim. // add tiago 31/01/2022
END_VAR
VAR_OUTPUT
	xHeartBeatSaida		: BOOL; // saida do Heart Beat pra ja ficar pornto no bloco né
	sTextoIMG 			: STRING; // saida para a imagem do coração
	xAlive 				: BOOL; // se esta conectado
	xDead 				: BOOL; // se nao esta conectado
END_VAR
VAR
	rtHeartBeatEntrada: R_TRIG;
	ftHeartBeatEntrada: F_TRIG;
	tonWatchDogEntrada: TON;
	xAliveEntrada : BOOL;
	
	tonHBSaida : TON;
	
END_VAR


IF xLicensaValida87208720 THEN
	

// Codigo criado por Ricardo Gajardo
// Transformado em function block por Tiago Bortolini Cunico em 27/08/2020
// Atualizado em 22/01/2022 por Tiago para a comunicação EAP de rolandia
// Atualizado para olhar a nossa licensa em 24/06/2022 por Tiago
// Corrigido o status de alive em 29/11/2022 por Tiago


	rtHeartBeatEntrada(CLK:=xHeartBeatEntrada, Q=> );// trigers para saber se ele morreu
	ftHeartBeatEntrada(CLK:=xHeartBeatEntrada, Q=> );
	
	tonWatchDogEntrada(IN:= NOT(rtHeartBeatEntrada.Q OR ftHeartBeatEntrada.Q), PT:= tTempoAlive, Q=>, ET=>); // se estiver morto por mais de 3 segundos ai avisa que esta morto
	
	xDead := tonWatchDogEntrada.q OR uiQualidade > 0;
	
	IF (xTK2000) THEN
		
		IF xHeartBeatEntrada AND NOT xDead THEN // controle da imagem
				sTextoIMG := 'Images/HeartBeatVd.png';
			ELSIF NOT xHeartBeatEntrada AND NOT xDead THEN
				sTextoIMG := 'Images/HeartBeatPt.png';
			ELSE
				sTextoIMG := 'Images/HeartBeatCz.png';			
		END_IF
		
	
	ELSE
	
		IF xHeartBeatEntrada AND NOT xDead THEN // controle da imagem
				sTextoIMG := 'HeartBeatVd';
			ELSIF NOT xHeartBeatEntrada AND NOT xDead THEN
				sTextoIMG := 'HeartBeatPt';
			ELSE
				sTextoIMG := 'HeartBeatCz';			
		END_IF
		
	END_IF
	
	xAlive := NOT xDead;
	
	tonHBSaida.IN := TRUE;
	IF tonHBSaida.q THEN
		xHeartBeatSaida := NOT xHeartBeatSaida;
		tonHBSaida.IN := FALSE;
	END_IF
	
	
	tonHBSaida(IN:= , PT:=T#100MS , Q=> , ET=> );

ELSE
	ValidaLicensa();
END_IF

END_FUNCTION_BLOCK

// FBs/EAP/FB_HarmonizaVariavel_Bool
FUNCTION_BLOCK FB_HarmonizaVariavel_Bool
VAR_IN_OUT
	Entrada_From : BOOL;
	Controle : BOOL;
	Saida_to : BOOL;
END_VAR
VAR_OUTPUT
END_VAR
VAR
	

	rtMudouVar1  : R_TRIG;
	var1Anterior : BOOL;
	
	rtMudouVar2  : R_TRIG;
	var2Anterior : BOOL;

END_VAR

IF xLicensaValida87208720 THEN
	
	
	rtMudouVar1(CLK:= Entrada_From <> var1Anterior, Q=> );
	IF rtMudouVar1.q THEN
		Controle := Entrada_From;
	END_IF
	var1Anterior := Entrada_From;
	
	
	rtMudouVar2(CLK:= Controle <> var2Anterior, Q=> );
	IF rtMudouVar2.q THEN
		Saida_to := Controle;
	END_IF
	var2Anterior := Controle;

ELSE
	ValidaLicensa();
END_IF

END_FUNCTION_BLOCK

// FBs/EAP/FB_HarmonizaVariavel_Int
FUNCTION_BLOCK FB_HarmonizaVariavel_Int
VAR_IN_OUT
	Entrada_From : INT;
	Controle : INT;
	Saida_to : INT;
END_VAR
VAR_OUTPUT
END_VAR
VAR
	
	rtMudouVar1  : R_TRIG;
	var1Anterior : INT;
	rtMudouVar2  : R_TRIG;
	var2Anterior : int;

END_VAR

IF xLicensaValida87208720 THEN
	

	rtMudouVar1(CLK:= Entrada_From <> var1Anterior, Q=> );
	IF rtMudouVar1.q THEN
		Controle := Entrada_From;
	END_IF
	var1Anterior := Entrada_From;
	
	
	rtMudouVar2(CLK:= Controle <> var2Anterior, Q=> );
	IF rtMudouVar2.q THEN
		Saida_to := Controle;
	END_IF
	var2Anterior := Controle;
ELSE
	ValidaLicensa();
END_IF

END_FUNCTION_BLOCK

// FBs/EAP/FB_HarmonizaVariavel_Real
FUNCTION_BLOCK FB_HarmonizaVariavel_Real
VAR_IN_OUT
	Entrada_From : REAL;
	Controle : REAL;
	Saida_to : REAL;
END_VAR
VAR_OUTPUT
END_VAR
VAR
	rtMudouVar1  : R_TRIG;
	var1Anterior : REAL;
	rtMudouVar2  : R_TRIG;
	var2Anterior : REAL;

END_VAR


IF xLicensaValida87208720 THEN
	
	rtMudouVar1(CLK:= Entrada_From <> var1Anterior, Q=> );
	IF rtMudouVar1.q THEN
		Controle := Entrada_From;
	END_IF
	var1Anterior := Entrada_From;
	
	
	rtMudouVar2(CLK:= Controle <> var2Anterior, Q=> );
	IF rtMudouVar2.q THEN
		Saida_to := Controle;
	END_IF
	var2Anterior := Controle;

ELSE
	ValidaLicensa();
END_IF

END_FUNCTION_BLOCK

// FBs/Diagnostico/KPI/FB_KPI_Geral
FUNCTION_BLOCK FB_KPI_Geral
VAR_INPUT
	xEstado1		: BOOL;
	sCorEstado1		: STRING;// cor em Hexa que vai aparecer no grafico de pizza na IHM
	sTextoEstado1 	: STRING; // texto que vai ser o titulo do estado 1 no grafico de pizza
	
	xEstado2		: BOOL;
	sCorEstado2		: STRING;// cor em Hexa que vai aparecer no grafico de pizza na IHM
	sTextoEstado2 	: STRING; // texto que vai ser o titulo do estado 1 no grafico de pizza
	
	sCorEstado3		: STRING;// cor em Hexa que vai aparecer no grafico de pizza na IHM
	sTextoEstado3 	: STRING; // texto que vai ser o titulo do estado 1 no grafico de pizza
	
	stHoraAgora		: TIMESTRUCT;
	
END_VAR
VAR_OUTPUT
	KPI : ARRAY[0..23] OF st_KPI_Geral;
END_VAR
VAR
	wSegAnterior	: WORD;
	whoraAnterior	: WORD;
	KPIVazio		: st_KPI_Geral;
	i				: INT;
	xFirstScan 		: BOOL := TRUE;
END_VAR

IF xLicensaValida87208720 THEN
	
	
	IF xFirstScan THEN
		FOR i := 0 TO 23 DO
			KPI[i].stGraficoIHM[0].x := sTextoEstado1;
			IF sCorEstado1 <> '' THEN
				KPI[i].stGraficoIHM[0].sCor := sCorEstado1;
			ELSE
				KPI[i].stGraficoIHM[0].sCor := '#555555';
			END_IF
			
			KPI[i].stGraficoIHM[1].x := sTextoEstado2;
			IF sCorEstado1 <> '' THEN
				KPI[i].stGraficoIHM[1].sCor := sCorEstado2;
			ELSE
				KPI[i].stGraficoIHM[1].sCor := '#F1F1F1';
			END_IF
			
			KPI[i].stGraficoIHM[2].x := sTextoEstado3;
			IF sCorEstado1 <> '' THEN
				KPI[i].stGraficoIHM[2].sCor := sCorEstado3;
			ELSE
				KPI[i].stGraficoIHM[2].sCor := '#FFFF00';
			END_IF
			
		END_FOR
	END_IF
	
	
	
	IF wSegAnterior <> stHoraAgora.wSecond THEN
	
		IF xEstado1 THEN
			KPI[0].rPorcEstado1	:= KPI[0].rPorcEstado1 + 0.027777;
			KPI[0].tEstado1		:= KPI[0].tEstado1 + T#1S;
		ELSIF xEstado2 THEN
			KPI[0].rPorcEstado2	:= KPI[0].rPorcEstado2 + 0.027777;
			KPI[0].tEstado2		:= KPI[0].tEstado2 + T#1S;
		END_IF
	
		KPI[0].rPorcEstado3 :=
			100 - KPI[0].rPorcEstado1 - KPI[0].rPorcEstado2;
	
		KPI[0].tEstado3 :=
			T#1H - KPI[0].tEstado1 - KPI[0].tEstado2;
	
	END_IF
	
	IF whoraAnterior <> stHoraAgora.wHour THEN
		FOR i := 23 TO 1 BY -1 DO
			KPI[i] := KPI[i - 1];
		END_FOR
		KPI[0] := kpiVazio;
	END_IF
	
	whoraAnterior	:= stHoraAgora.wHour;
	wSegAnterior	:= stHoraAgora.wSecond;
	
	
	
	
	xFirstScan := TRUE;

END_IF

END_FUNCTION_BLOCK

// FBs/Emergencia/FB_Emergencia
FUNCTION_BLOCK FB_Emergencia
VAR_IN_OUT
	stEmergencia : st_Emergencia;
END_VAR
VAR_INPUT
	xEmergenciaOK : BOOL; // status da emergencia, se for externa tb serve
	sNomeFuncao : STRING;
	xControleTCSafe : BOOL;
	xControleInterno : BOOL;
	xCH1 : BOOL;
	xCH2 : BOOL;
	xbypassCH2 : BOOL;
	tDiscrepancia : TIME;
	xReset : BOOL;
	xResetFisico : BOOL;
	stHoraAgora : TIMESTRUCT;
END_VAR
VAR_OUTPUT
	kpi : ARRAY[0..23] OF st_KPI_Geral;
	xErro : BOOL;
	xLedReset : BOOL;
	sEstadoIHM : STRING;
	iEstado : INT;//0 : desligado, 1 : OK, 2 : Esperando Reset, 3 : Desincronizado, 4 : EDM, 5 : Outro Erro
END_VAR
VAR
	tonDiscrepencia : TON;
	wSegAnterior 	: WORD;
	wHoraAnterior 	: WORD;
	kpiVazio		: st_KPI_Geral;
	
	xFirstScan : BOOL := TRUE;
	
	i : INT;
	
	fbTNFDiscrepancia : FB_TimerOnOff;
	fbTNFAcionada : FB_TimerOnOff;
	
	{attribute 'tc_no_symbol'}
	{attribute 'hide'}
	stEmergenciaAnterior : st_Emergencia;
	
	xErroGrupo : BOOL;
	xSafeOut : BOOL;
	xSafetyOn : BOOL;
	xSafetyError : BOOL;
	
	xT20004000 : BOOL;	
	tonT20004000 : FB_TimerOnOff;
	xT200 : BOOL;	
	tonT200 : ton;
	xT1000 : BOOL;
	tonT1000 : ton;
	
END_VAR


IF xLicensaValida87208720 THEN
		
	
	
	IF xFirstScan THEN
		FirstScan();
	END_IF
	
	AjeitaEntrada();
	
	Timers();
	
	IF NOT stEmergencia.Config.xControleTCSafe THEN
	
		IF xControleInterno THEN
			IF xbypassCH2 THEN
				xCH2 := xCH1;
			END_IF
				
			IF ( NOT xCH1 OR NOT xCH2) OR tonDiscrepencia.q THEN
				xEmergenciaOK := FALSE;
			END_IF
			
			tonDiscrepencia(IN:= (xCH1 <> (xCH2)) AND NOT xErro, PT:= tDiscrepancia, Q=> , ET=> );
			IF tonDiscrepencia.q THEN
				xErro := TRUE;
			END_IF
			
			IF xReset OR xResetFisico THEN
				xErro := FALSE;
				xEmergenciaOK := TRUE;
				xReset := FALSE;
				xResetFisico := FALSE;
			END_IF
		ELSE
			xCH2 := xCH1 := xEmergenciaOK;
			xErro := FALSE;
		END_IF
		

		
		fbTNFDiscrepancia(
			xEnabled:= TRUE, 
			xLiga:= NOT xEmergenciaOK, 
			tON:= T#500MS, 
			tOF:= T#500MS, 
			xAciona=> xLedReset, 
			tTempoAteOProximoAcionamento=> );
			
		fbTNFAcionada(
			xEnabled:= TRUE, 
			xLiga:= xErro, 
			tON:= T#250MS, 
			tOF:= T#250MS, 
			xAciona=> , 
			tTempoAteOProximoAcionamento=> );
		
		
		IF xErro THEN
			xLedReset := fbTNFAcionada.xAciona;
		END_IF
	
	ELSE // Safety beckhoff
		
	
		stEmergencia.Safe.RESET := xReset OR xResetFisico;
		stEmergencia.Safe.ERRACK := xReset OR xResetFisico;
		stEmergencia.Safe.RUN := TRUE;


		CASE stEmergencia.Safe.State OF
			
			1: // OK
				xLedReset := FALSE;
				xEmergenciaOK := TRUE;
			
			2,4: // Discrepancia ou erro
				(* aceso por 2s, pisca por 4s *)
				IF xT20004000 THEN
					xLedReset := TRUE;
				ELSE
					xLedReset := xT200;
				END_IF
				xEmergenciaOK := FALSE;
				
			
			3: // Precionada
			
				xLedReset := xT1000;			(* pisca a cada 1s *)
				
				xEmergenciaOK := FALSE;
				
		ELSE
			
			xLedReset := FALSE;
			
		END_CASE
			

	END_IF
	
	CalculaKPIs();
	
	AjeitaSaida();
	
	xFirstScan := FALSE;
	

ELSE
	//ValidaLicensa();
END_IF

ACTION AjeitaEntrada:


IF stEmergencia.Config.tDiscrepancia <> stEmergenciaAnterior.Config.tDiscrepancia THEN
	tDiscrepancia := stEmergencia.Config.tDiscrepancia;
END_IF
IF stEmergencia.Config.tDiscrepancia <> tDiscrepancia THEN
	stEmergencia.Config.tDiscrepancia := tDiscrepancia;
END_IF

IF stEmergencia.Config.xbypassCH2 <> stEmergenciaAnterior.Config.xbypassCH2 THEN
	xbypassCH2 := stEmergencia.Config.xbypassCH2;
END_IF
IF stEmergencia.Config.xbypassCH2 <> xbypassCH2 THEN
	stEmergencia.Config.xbypassCH2 := xbypassCH2;
END_IF

IF stEmergencia.Config.xControleInterno <> stEmergenciaAnterior.Config.xControleInterno THEN
	xControleInterno := stEmergencia.Config.xControleInterno;
END_IF
IF stEmergencia.Config.xControleInterno <> xControleInterno THEN
	stEmergencia.Config.xControleInterno := xControleInterno;
END_IF

IF stEmergencia.En.xReset <> stEmergenciaAnterior.En.xReset THEN
	xReset := stEmergencia.En.xReset;
END_IF
IF stEmergencia.En.xReset <> xReset THEN
	stEmergencia.En.xReset := xReset;
END_IF

IF stEmergencia.En.xEmergenciaOK <> stEmergenciaAnterior.En.xEmergenciaOK THEN
	xEmergenciaOK := stEmergencia.En.xEmergenciaOK;
END_IF
IF stEmergencia.En.xEmergenciaOK <> xEmergenciaOK THEN
	stEmergencia.En.xEmergenciaOK := xEmergenciaOK;
END_IF

IF stEmergencia.En.xResetFisico <> stEmergenciaAnterior.En.xResetFisico THEN
	xResetFisico := stEmergencia.En.xResetFisico;
END_IF
IF stEmergencia.En.xResetFisico <> xResetFisico THEN
	stEmergencia.En.xResetFisico := xResetFisico;
END_IF




xCH1 := stEmergencia.En.xCH1;
xCH2 := stEmergencia.En.xCH2; 









stEmergenciaAnterior := stEmergencia;
END_ACTION

ACTION AjeitaSaida:


stEmergencia.Sa.kpi := kpi;
stEmergencia.Sa.xErro := xErro;
stEmergencia.Sa.xLedReset := xLedReset;

stEmergencia.En.sNomeFuncao := sNomeFuncao := CONCAT(CONCAT(stemergencia.Banco.Tag,' - '),stemergencia.Banco.Funcao);

IF NOT stEmergencia.Config.xControleTCSafe THEN
	
	
	IF xErro THEN
		sEstadoIHM := 'Discrepancia';
		iEstado := 3;
	ELSIF NOT xCH1 THEN
		sEstadoIHM := 'Esperando Reset';
		iEstado := 3;
	ELSIF NOT xEmergenciaOK THEN
		sEstadoIHM := 'Esperando Reset';
		iEstado := 2;
	END_IF
	
	IF xEmergenciaOK THEN
		sEstadoIHM := 'OK';
		iEstado := 1;
	END_IF
ELSE
	
	CASE stEmergencia.Safe.State OF
		0:
			sEstadoIHM := 'Offline';
			iEstado := 0;
		1 :
			sEstadoIHM := 'OK';
			iEstado := 1;
		2:
			sEstadoIHM := 'FB em STOP ';
			iEstado := 5;
		3:
			sEstadoIHM := 'Emergencia pressionada ';
			iEstado := 2;
		4:
			sEstadoIHM := 'Erro ';
			iEstado := 5;
		5:
			sEstadoIHM := 'FB em RESET ';
			iEstado := 5;
		6:
			sEstadoIHM := 'FB em START';
			iEstado := 5;
		8:
			sEstadoIHM := 'FB em DELAYOUT ';
			iEstado := 5;
	END_CASE
	
	IF (stEmergencia.Safe.Diag AND 2#0000000000000001) > 0 THEN
		sEstadoIHM := CONCAT(sEstadoIHM,'| Discrepancia G1 ');
		iEstado := 3;
	END_IF
	IF (stEmergencia.Safe.Diag AND 2#0000000000000010) > 0 THEN
		sEstadoIHM := CONCAT(sEstadoIHM,'| Discrepancia G2 ');
		iEstado := 3;
	END_IF
	IF (stEmergencia.Safe.Diag AND 2#0000000000000100) > 0 THEN
		sEstadoIHM := CONCAT(sEstadoIHM,'| Discrepancia G3 ');
		iEstado := 3;
	END_IF
	IF (stEmergencia.Safe.Diag AND 2#0000000000001000) > 0 THEN
		sEstadoIHM := CONCAT(sEstadoIHM,'| Discrepancia G4 ');
		iEstado := 3;
	END_IF
	IF (stEmergencia.Safe.Diag AND 2#0000000000010000) > 0 THEN
		sEstadoIHM := CONCAT(sEstadoIHM,'| EDM 1 ');
		iEstado := 4;
	END_IF
	IF (stEmergencia.Safe.Diag AND 2#0000000000100000) > 0 THEN
		sEstadoIHM := CONCAT(sEstadoIHM,'| EDM 2 ');
		iEstado := 4;
	END_IF
	
END_IF

stEmergencia.Sa.sEstadoIHM := sEstadoIHM;

stEmergencia.Sa.iStatus := iEstado;
END_ACTION

ACTION CalculaKPIs:


IF wSegAnterior <> stHoraAgora.wSecond THEN

	IF NOT xEmergenciaOK THEN
		KPI[0].rPorcEstado2	:= KPI[0].rPorcEstado2 + 0.027777;
		KPI[0].tEstado2		:= KPI[0].tEstado2 + T#1S;
	END_IF


	KPI[0].rPorcEstado1 := 100 - KPI[0].rPorcEstado2;
	KPI[0].tEstado1 := T#1H - KPI[0].tEstado2;
		

	KPI[0].stGraficoIHM[0].y := KPI[0].rPorcEstado1;
	KPI[0].stGraficoIHM[1].y := KPI[0].rPorcEstado2;
	

END_IF

IF whoraAnterior <> stHoraAgora.wHour THEN
	FOR i := 23 TO 1 BY -1 DO
		KPI[i] := KPI[i - 1];
	END_FOR

	KPI[0] := kpiVazio;
	
	KPI[0].stGraficoIHM[0].x := 'OK';
	KPI[0].stGraficoIHM[0].sCor := '#555555';
	
	KPI[0].stGraficoIHM[1].x := 'Acionada';
	KPI[0].stGraficoIHM[1].sCor := '#FF0000';
END_IF

whoraAnterior	:= stHoraAgora.wHour;
wSegAnterior	:= stHoraAgora.wSecond;
END_ACTION

ACTION FirstScan:

stEmergenciaAnterior := stEmergencia;

whoraAnterior	:= stHoraAgora.wHour;
wSegAnterior	:= stHoraAgora.wSecond;


FOR i := 0 TO 23 DO
	KPI[i].stGraficoIHM[0].x := 'OK';
	KPI[i].stGraficoIHM[0].sCor := '#555555';
	KPI[i].stGraficoIHM[0].y := 100;
	
	KPI[i].stGraficoIHM[1].x := 'Acionada';
	KPI[i].stGraficoIHM[1].sCor := '#FF0000';
END_FOR
END_ACTION

ACTION Timers:

tonT20004000(
	xEnabled:= TRUE, 
	xLiga:= TRUE, 
	tON:= T#2S, 
	tOF:= T#4S, 
	xAciona=> xT20004000, 
	tTempoAteOProximoAcionamento=> );



IF tonT200.q THEN
	xT200 := NOT xT200;
	tonT200(IN:= FALSE, PT:=T#200MS);
END_IF
tonT200(IN:= TRUE, PT:=T#200MS);


IF tonT1000.q THEN
	xT1000 := NOT xT1000;
	tonT1000(IN:= FALSE, PT:=T#1000MS);
END_IF
tonT1000(IN:= TRUE, PT:=T#1000MS);
END_ACTION

END_FUNCTION_BLOCK

// FBs/Controle/FB_TimerOnOff
FUNCTION_BLOCK FB_TimerOnOff
VAR_INPUT
	xEnabled : BOOL;
	xLiga : BOOL;
	tON : TIME;
	tOF : TIME;
END_VAR
VAR_OUTPUT
	xAciona : BOOL;
	tTempoAteOProximoAcionamento : TIME;
END_VAR
VAR
	tonOF : TON;
	tonON : TON;
	rtLiga : R_TRIG;
	ftDesliga : F_TRIG;
	xLigado : BOOL;
	xInicia_tonOF : BOOL;
END_VAR

IF xLicensaValida87208720 THEN
//Criado por Tiago Bortolini Cunico
	
	
	IF xEnabled THEN
		
		rtLiga(CLK:= xLiga, Q=> );// inicia a contagem
		IF rtLiga.q THEN
			xLigado := TRUE;
			xInicia_tonOF := TRUE;
		END_IF
		
		ftDesliga(CLK:= xLiga, Q=> );// para tudo
		IF ftDesliga.q THEN
			xLigado := FALSE;
			xInicia_tonOF := FALSE;
			xAciona := false;
		END_IF
		
	
			
		tonOF(IN:= xInicia_tonOF AND xLigado, PT:= tOF, Q=> , ET=> );
		
		
		
		IF tonOF.Q THEN
			xInicia_tonOF := FALSE;
			xAciona := TRUE;
		END_IF
	
		tonON(IN:= NOT xInicia_tonOF AND xLigado, PT:= tON, Q=> , ET=> );
		
		IF tonON.Q THEN
			xInicia_tonOF := TRUE;
			xAciona := FALSE;
		END_IF
		
	
		IF xAciona THEN
			tTempoAteOProximoAcionamento := TON - tonON.ET;
		ELSE
			tTempoAteOProximoAcionamento := tOF - tonOF.ET;
		END_IF
	
END_IF	





































































ELSE
	ValidaLicensa();
END_IF

END_FUNCTION_BLOCK

// FBs/Alarmes/GerenciadorV2/FB_GerenciadorAlarmesV2
{attribute 'hide_all_locals'}
FUNCTION_BLOCK FB_GerenciadorAlarmesV2
VAR_IN_OUT
	Alarmes_Array		: ARRAY[*] OF ST_Alarmes_V2;			//Array com os Dados para Tabela de Alarme Online
	Alarmes_Online		: ARRAY[*] OF ST_Alarmes_Online_V2;		//Array com os Dados para Tabela de Alarme Online
	Alarmes_Historico	: ARRAY[0..1000] OF ST_Alarmes_Historico_V2;	//Array com os Dados para Tabela de Alarme Histórico
	RT					: ARRAY[*] OF R_TRIG;					//
	FT					: ARRAY[*] OF F_TRIG;					//
END_VAR
VAR_INPUT
	xReconheceAlarmes	: BOOL;
	sData				: STRING;
	sHora				: STRING;
	sUser				: STRING;
	iMaxIteracao		: INT := 10;
END_VAR
VAR_OUTPUT
	xAlarmeAtivo			: BOOL;
	xAlarmeAtivoReconhecido	: BOOL;
END_VAR
VAR
	iMin	: UDINT;
	iMax	: UDINT;

	iMaxHistorico : INT := 1000;

	pFT	: POINTER TO BOOL;
	pRT	: POINTER TO BOOL;

	i			: INT;
	j			: INT;
	k			: INT;
	iContAcoes	: INT;
	xFirstScan	: BOOL := TRUE;

	AlarmeOnlineVazio : ST_Alarmes_Online_V2;
	iAux : INT;
	iAux2 : INT;
END_VAR

IF xLicensaValida87208720 THEN
	
	// 0 nao ativo
	// 1 ativo nao reconhecido
	// 2 reconhecido e ativo
	// 3 reconhecido e nao mais ativo
	// 4 off e nao foi reconhecido
	
	IF xFirstScan THEN
		//ve o tamanho max e min
		iMax			:= DINT_TO_UDINT(UPPER_BOUND(Alarmes_Array, 1));
		//iMaxHistorico	:= TO_INT(UPPER_BOUND(Alarmes_Historico, 1));
		(*
		// gera os ft e rt pra isso
		pRT	:= __NEW(BOOL, iMax);
		pFT	:= __NEW(BOOL, iMax);
		*)
	END_IF
	
	// passa em todos os alarmes ativos e joga pra reconhecido 
	IF xReconheceAlarmes THEN
		FOR i := 0 TO TO_INT(iMax) DO
			IF Alarmes_Online[i].sData <> '' THEN
				Alarmes_Online[i].iStatus := 2;
			ELSE
				EXIT;
			END_IF
	
		END_FOR
	END_IF
	
	iContAcoes := 0;
	FOR i := 0 TO TO_INT(iMax) DO
		// quando da borda de subida em um alarme ele sobe esse alarme
		RT[i](CLK := Alarmes_Array[i].xAtivo);
		IF RT[i].Q THEN
			SobeAlarme();
			iContAcoes := iContAcoes + 1;
		END_IF
	
		// quando da borda de descida em um alarme ele desce esse alarme
		FT[i](CLK := Alarmes_Array[i].xAtivo);
		IF FT[i].Q THEN
			DesceAlarme();
			iContAcoes := iContAcoes + 1;
		END_IF
		
		IF iContAcoes > iMaxIteracao THEN
			EXIT;
		END_IF
		
	END_FOR
	
	xAlarmeAtivo			:= FALSE;
	xAlarmeAtivoReconhecido	:= FALSE;
	
	FOR i := 0 TO TO_INT(iMax) DO
	
		xAlarmeAtivo			:= xAlarmeAtivo OR Alarmes_Online[i].iStatus = 1;
		xAlarmeAtivoReconhecido	:= xAlarmeAtivoReconhecido OR Alarmes_Online[i].iStatus = 2;
	
		IF Alarmes_Online[i].sHora = '' THEN
			EXIT;
		END_IF
	END_FOR
	
	xFirstScan := FALSE;

ELSE
	ValidaLicensa();
END_IF

ACTION DesceAlarme:

//codigo para quando um alarme desce para o historico

//joga todos os alarmes 1 pra tras
FOR j := TO_INT(iMaxHistorico - 1) TO 0 BY -1 DO
	Alarmes_Historico[j + 1] := Alarmes_Historico[j];
END_FOR

// ve qual alarme online é oq caiu pelo identificador
FOR j := 0 TO TO_INT(iMax) DO
	IF Alarmes_Online[j].iIdentificador = i THEN
		EXIT;
	END_IF
END_FOR

//coloca a data e a hora
Alarmes_Historico[0].sData_on := Alarmes_Online[j].sData;
Alarmes_Historico[0].sHora_on := Alarmes_Online[j].sHora;
Alarmes_Historico[0].iTipo    := Alarmes_Online[j].iTipo;
// se for alarme coloca fim
IF Alarmes_Historico[0].iTipo = 0 THEN
	Alarmes_Historico[0].sData_off := sData;
	Alarmes_Historico[0].sHora_off := sHora;
ELSE
	// se for mensagem ai nao precisa
	Alarmes_Historico[0].sData_off := sData;
	Alarmes_Historico[0].sHora_off := sHora;
END_IF

Alarmes_Historico[0].sTexto   := Alarmes_Online[j].sMensagem;
Alarmes_Historico[0].sUsuario := Alarmes_Online[j].sUser;
Alarmes_Historico[0].sTAG     := Alarmes_Online[j].sTAG;

IF Alarmes_Historico[0].iTipo = 0 THEN
	// se for alarme
	CASE Alarmes_Online[j].iStatus OF
		1:
			Alarmes_Historico[0].iStatus := 4;

		2:
			Alarmes_Historico[0].iStatus := 3;
	END_CASE
ELSE
	//se for mensagem
	Alarmes_Historico[0].iStatus := 5;
END_IF

// limpa o alarme que nao ta mais ativo
Alarmes_Online[j] := AlarmeOnlineVazio;

// puxa todos os alarmes de tras dele 1 pra frente
FOR k := j TO TO_INT(iMax - 1) DO
	// se for = '' é pq nao tem mais que puxar eles pra cima ai ele pula fora
	Alarmes_Online[k] := Alarmes_Online[k + 1];

	IF Alarmes_Online[k + 1].sMensagem = '' THEN
		EXIT;
	END_IF
END_FOR
END_ACTION

ACTION SobeAlarme:

//codigo para quando um alarme sobe para os onlines


(*
FOR iAux2 := 0 TO UDINT_TO_INT(iMax) DO
	IF Alarmes_Online[i].sHora <> '' THEN
		iAux := iAux2;
		EXIT;
	END_IF
END_FOR
*)

//joga todos os alarmes 1 pra tras
FOR j := UDINT_TO_INT(iMax - 1) TO 0 BY -1 DO
	Alarmes_Online[j + 1] := Alarmes_Online[j];
END_FOR

//coloca a data e a hora
Alarmes_Online[0].sData          := sData;
Alarmes_Online[0].sHora          := sHora;
Alarmes_Online[0].iStatus        := 1;
Alarmes_Online[0].sUser          := sUser;
Alarmes_Online[0].sTAG           := Alarmes_Array[i].sTAG;
Alarmes_Online[0].iTipo          := Alarmes_Array[i].iTipo;
Alarmes_Online[0].sMensagem      := Alarmes_Array[i].sTexto;
Alarmes_Online[0].iIdentificador := i;
END_ACTION

END_FUNCTION_BLOCK

// FBs/Alarmes/GerenciadorV2/Mensagens/FB_MensagemMudouBool
FUNCTION_BLOCK FB_MensagemMudouBool
VAR_IN_OUT
	stAlarme : ST_Alarmes_V2;
END_VAR
VAR_INPUT
	xBool : BOOL;
END_VAR
VAR_OUTPUT
	xMudou        : BOOL;
	xboolAnterior : BOOL;
END_VAR
VAR
	rtTaDiferente : R_TRIG;
	xFirstScan : BOOL := TRUE;
END_VAR


IF xFirstScan THEN
	xboolAnterior := xBool;
	xFirstScan := FALSE;
END_IF


stAlarme.xAtivo := FALSE;
stAlarme.iTipo  := 1;

rtTaDiferente(CLK := xboolAnterior <> xBool, Q =>);

IF rtTaDiferente.q THEN
	stAlarme.xAtivo := TRUE;
END_IF

xMudou := stAlarme.xAtivo;
xboolAnterior := xBool;

END_FUNCTION_BLOCK

// FBs/Alarmes/GerenciadorV2/Mensagens/FB_MensagemMudouInt
FUNCTION_BLOCK FB_MensagemMudouInt
VAR_IN_OUT
	stAlarme : ST_Alarmes_V2;
END_VAR
VAR_INPUT
	iInt    : INT;
END_VAR
VAR_OUTPUT
	xMudou : BOOL;
	iIntAnterior : INT;
END_VAR
VAR
	rtTaDiferente : R_TRIG;
	xFirstScan : BOOL := TRUE;
END_VAR


IF xFirstScan THEN
	iIntAnterior := iInt;
	xFirstScan := FALSE;
END_IF

stAlarme.xAtivo := FALSE;
stAlarme.iTipo  := 1;

rtTaDiferente(CLK := iIntAnterior <> iInt, Q =>);

IF rtTaDiferente.q THEN
	stAlarme.xAtivo := TRUE;
ELSE
	iIntAnterior := iInt;
END_IF

xMudou := stAlarme.xAtivo;

END_FUNCTION_BLOCK

// FBs/Alarmes/GerenciadorV2/Mensagens/FB_MensagemMudouReal
FUNCTION_BLOCK FB_MensagemMudouReal
VAR_IN_OUT
	stAlarme : ST_Alarmes_V2;
END_VAR
VAR_INPUT
	rReal    : REAL;
END_VAR
VAR_OUTPUT
	xMudou : BOOL;
	rRealAnterior : REAL;
END_VAR
VAR
	rtTaDiferente : R_TRIG;
	xFirstScan : BOOL := TRUE;
END_VAR



IF xFirstScan THEN
	rRealAnterior := rReal;
	xFirstScan := FALSE;
END_IF


stAlarme.xAtivo := FALSE;
stAlarme.iTipo  := 1;

rtTaDiferente(CLK := rRealAnterior <> rReal, Q =>);

IF rtTaDiferente.q THEN
	stAlarme.xAtivo := TRUE;
ELSE
	rRealAnterior := rReal;
END_IF

xMudou := stAlarme.xAtivo;

END_FUNCTION_BLOCK

// FBs/Controle/BotaoDeParada/FB_BotaoParada
FUNCTION_BLOCK FB_BotaoParada
VAR_INPUT
	xSinalBP		: BOOL;
END_VAR
VAR_OUTPUT
	xParadaAcionada	: BOOL := FALSE;
	xLedBotao		: BOOL;
END_VAR
VAR
	rtBotao		: Tc2_Standard.R_TRIG;
	tonPiscaLed	: Tc2_Standard.TON;
	xPisca		: BOOL;
END_VAR


IF xLicensaValida87208720 THEN

	rtBotao(CLK:= xSinalBP, Q=> );
	
	IF rtBotao.Q THEN
		xParadaAcionada := NOT xParadaAcionada;
	END_IF
	
	tonPiscaLed(IN:= TRUE, PT:= T#1S, Q=> , ET=> );
	
	IF tonPiscaLed.Q THEN
		tonPiscaLed(IN:= FALSE, PT:= T#1S, Q=> , ET=> );
		xPisca := NOT xPisca;
	END_IF
	
	
	xLedBotao := xParadaAcionada AND xPisca;
		
ELSE
	ValidaLicensa();
END_IF

END_FUNCTION_BLOCK

// FBs/Controle/Telerruptor/FB_IniciaOsBlocosDeConfigDoTelerruptor
FUNCTION_BLOCK FB_IniciaOsBlocosDeConfigDoTelerruptor
VAR_IN_OUT
	stTelerruptor		: ARRAY[*] OF stTelerruptor;
END_VAR
VAR_INPUT
	xInicia			: BOOL;
	xCriaTabela		: BOOL;
	iNumeroDataBase	: INT		:= 1;
	sNomeDataBase	: STRING	:= 'iluminacaoconfig';
END_VAR
VAR_OUTPUT
	xOcupado	: BOOL;
END_VAR
VAR
	
	//Cria table
	rtCria			: R_TRIG;
	xCria			: BOOL;
	fbPLCDBCreate	: FB_PLCDBCreateEvt(sNetID := '', tTimeout := T#30S);
	ColumnInfo : ARRAY[0..2] OF ST_ColumnInfo := [(sName := 'Telerruptor', eType := E_ColumnType.Integer, nLength := 8, sProperty := 'IDENTITY(1,1)'),
												  (sName := 'Tag', eType := E_ColumnType.NVarChar, nLength := 80, sProperty := 'DEFAULT $'SEMTAG$''),
												  (sName := 'Funcao', eType := E_ColumnType.NVarChar, nLength := 80, sProperty := 'DEFAULT $'NADA$'')];
												  
												  
	//Gera os Telerruptores
	diParteBaixa		: DINT;
	diParteAlta			: DINT;
	i					: INT;
	j					: INT;
	xGeraTelerruptores	: BOOL;
	xEscreve			: BOOL;
	xEscreveAux			: BOOL;
	rtEscrita			: R_TRIG;	
	EstruturaBanco		: ARRAY[0..999] OF ConfigTelerruptorDB;
	fbPLCDBWrite		: FB_PLCDBWriteEvt(sNetID := '', tTimeout := T#30S); //Bloco para gravar no banco de dados
	ColumnNamesGrava	: ARRAY[0..2] OF STRING(50) := ['Telerruptor',
														'Tag',
														'Funcao'
														];
														
														
	//Le os nomes
	xFirstScan		: BOOL := TRUE;
	xLe				: BOOL;
	sCmd			: STRING(1000);
	sTag1			: STRING;
	TagAProcurar	: STRING(80);
	sMensagemErro1	: STRING;
	iIndexGrava		: INT := 0;
	iAux			: DINT;
	diCima			: DINT;
	diBaixo			: DINT;
	nRecords		: UDINT;
	Anterior		: ARRAY[0..999] OF stTelerruptor;
	stPara			: ST_ExpParameter;
	EstruturaBancoLe: ARRAY[0..999] OF ConfigTelerruptorDB;
	eEstado			: enum_LeituradosNomes := enum_LeituradosNomes.eEsperando;
	fbSQLDatabase	: FB_SQLDatabaseEvt(sNetID := '', tTimeout := T#30S);
	fbPLCDBCmd		: FB_PLCDBCmdEvt(sNetID := '', tTimeout := T#30S);
	
	//Grava Nomes Novos
	xGrava			: BOOL;
	xAberto			: BOOL;
	sCmd2			: STRING(1000);
	sMensagemErro2	: STRING;
	Nome			: STRING;
	Vazio			: STRING := '';
	Tag				: STRING;
	Funcao			: STRING;
	arrStr			: ARRAY[1..10] OF STRING(255);
	eEstadoGrava	: enum_GravaNomes := enum_GravaNomes.eEsperando;
	fbSqlCommand		: FB_SQLCommandEvt(sNetID := '', tTimeout := T#30S);
	fbSQLDatabase2	: FB_SQLDatabaseEvt(sNetID := '', tTimeout := T#30S);

END_VAR


IF xFirstScan THEN
	xLe := TRUE;
	//xCriaTabela := TRUE;
END_IF

IF xInicia THEN
	xLe := TRUE;
	eEstado := enum_LeituradosNomes.eEsperando;
END_IF

GeraTabela();
GeraOsTelerruptores();
LeNomes();
GravaValores();


xFirstScan	:= FALSE;
xInicia		:= FALSE;

ACTION GeraOsTelerruptores:

diParteBaixa	:= LOWER_BOUND(stTelerruptor, 1);
diParteAlta		:= UPPER_BOUND(stTelerruptor, 1);

IF xGeraTelerruptores THEN

	xEscreve := TRUE;
	rtEscrita(CLK := xEscreve, Q =>);

	IF rtEscrita.q THEN
		xEscreveAux						:= TRUE;
		xOcupado						:= TRUE;
		j := DINT_TO_INT(diParteBaixa) + 1;
	END_IF

	IF xEscreveAux THEN
		EstruturaBanco[j].Tag := CONCAT('IL', INT_TO_STRING(j));
		EstruturaBanco[j].Telerruptor := INT_TO_DINT(j);
		
		IF fbPLCDBWrite.WriteStruct
		(
			hDBID := INT_TO_UDINT(iNumeroDataBase),
				sTableName := sNomeDataBase,
				pRecord := ADR(EstruturaBanco[j]),
				cbRecord := SIZEOF(EstruturaBanco[j]),
				pColumnNames := ADR(ColumnNamesGrava),
				cbColumnNames := SIZEOF(ColumnNamesGrava))
		THEN
			j := j +1;
		ELSE
			IF fbPLCDBWrite.bError THEN
				IF fbPLCDBWrite.ipTcResult.nEventId = 61 THEN
					xCriaTabela := TRUE;
				END_IF
			END_IF
		END_IF
		
		IF j > diParteAlta THEN
			xOcupado	:= FALSE;
			xEscreve 	:= FALSE;
			rtEscrita(CLK := xEscreve, Q =>);
			xEscreveAux	:= FALSE;
			xGeraTelerruptores := FALSE;
			j := DINT_TO_INT(diParteBaixa);
			
			xLe := TRUE;
			eEstado := enum_LeituradosNomes.eEsperando;
		END_IF

	END_IF
END_IF
END_ACTION

ACTION GeraTabela:

rtCria(CLK := xCriaTabela, Q =>);

IF rtCria.q THEN
	xCria		:= TRUE;
	xOcupado	:= TRUE;
END_IF

IF xCria THEN

	IF fbPLCDBCreate.Table
		(
			hDBID := INT_TO_UDINT(iNumeroDataBase),
				sTableName := sNomeDataBase,
				pTableCfg := ADR(ColumnInfo),
				cbTableCfg := SIZEOF(ColumnInfo))
	THEN
		xCria		:= FALSE;
		xCriaTabela	:= FALSE;
		xOcupado	:= FALSE;
		xGeraTelerruptores	:= TRUE;
		j			:= 1;
	END_IF

END_IF
END_ACTION

ACTION GravaValores:
CASE eEstadoGrava OF
		enum_GravaNomes.eEsperando: //Esperando
			IF xGrava THEN
				IF xAberto THEN
					eEstadoGrava := enum_GravaNomes.eCriaComando;
				ELSE
					eEstadoGrava := enum_GravaNomes.eAbreConexao;
				END_IF
				
			END_IF
			
		enum_GravaNomes.eAbreConexao: //abre conexao
			IF fbSQLDatabase2.Connect(INT_TO_UDINT(iNumeroDataBase)) THEN
				IF fbSQLDatabase2.bError THEN
					{error <'Não conseguiu abrir a conexao no banco do bloco FB_IniciaOsBlocosDeConfigDoMotor 1'>}
					IF fbSQLDatabase2.ipTcResult.ipSourceInfo.sName = 'ADSERR_DEVICE_LICENSENOTFOUND' THEN
						// se der isso ele nao fica tentando e gerando uma caralhada de erro pq nao tem a lisença
						eEstadoGrava := enum_GravaNomes.eParado;
					ELSE
						eEstadoGrava := enum_GravaNomes.eAbreConexao;
					END_IF
					
				ELSE
					IF fbSQLDatabase2.bConnected THEN
						eEstadoGrava := enum_GravaNomes.eCriaComando;
						xAberto := TRUE;
					ELSE
						eEstadoGrava := enum_GravaNomes.eFechaConexao;
						xAberto := FALSE;
					END_IF
				END_IF
			END_IF
			
		enum_GravaNomes.eCriaComando:
			IF fbSQLDatabase2.CreateCmd(ADR(fbSqlCommand)) THEN
				IF fbSQLDatabase2.bError THEN
					eEstadoGrava := enum_GravaNomes.eCriaComando;
				ELSE
					eEstadoGrava := enum_GravaNomes.eGravaNomes;
				END_IF
			END_IF
			
		enum_GravaNomes.eGravaNomes:
	
			//UPDATE `geral`.`iluminacaoconfig` SET `Tag` = 'IL' WHERE (`Telerruptor` = '1');
			
			Nome := stTelerruptor[iIndexGrava].Config.sNome_Funcao;
			Tag := CONCAT(CONCAT('IL', TO_STRING(iIndexGrava)), ' - ');
		
			IF FindAndReplace(
						pSrcString:= ADR(Nome), 
						pDeleteString:= ADR(Tag), 
						pInsertString:= ADR(Vazio), 
						pDstString:= ADR(Funcao), 
						nDstSize:= SIZEOF(Funcao)) = 0  THEN
						
				Funcao := '';	
			END_IF
						
			arrStr[1] := 'UPDATE GERAL.';
			arrStr[2] := sNomeDataBase;
			arrStr[3] := ' SET Funcao = "';
			arrStr[4] := Funcao;
			arrStr[5] :='" WHERE (Telerruptor = "';
			arrStr[6] := TO_STRING(iIndexGrava);
			arrStr[7] := '");';
			
			sCmd2 := F_ConcatArray(sArray:= arrStr); 
	
			IF fbSQLCommand.Execute(pSQLCmd := ADR(sCmd2), cbSQLCmd := SIZEOF(sCmd2))
			THEN
				IF fbSQLCommand.bError THEN
					IF fbSQLCommand.ipTcResult.nEventId = 61 THEN
					// Esse erro acontece quando o database não tá criado, nesse caso ele tenta criar
						eEstadoGrava := enum_GravaNomes.eEsperando;
						xCriaTabela := TRUE;
					ELSE
						eEstadoGrava := enum_GravaNomes.eAbreConexao;
					END_IF
					sMensagemErro2 := 'Nao conseguiu a tag';
				ELSE
					sMensagemErro2	:= 'Conseguiu a tag';
				END_IF
				eEstadoGrava := enum_GravaNomes.eFechaConexao;
				iIndexGrava := 0;
			END_IF
			
		enum_GravaNomes.eFechaConexao:
			IF fbSQLDatabase2.Disconnect() THEN
		
				xGrava := FALSE;
				xLe := TRUE;
		
				IF fbSQLDatabase2.bError THEN
					eEstadoGrava := enum_GravaNomes.eEsperando;
				ELSE
					eEstadoGrava := enum_GravaNomes.eEsperando;
					xAberto := FALSE;
				END_IF
			END_IF

END_CASE
END_ACTION

ACTION LeNomes:

CASE eEstado OF
		enum_LeituradosNomes.eEsperando: //Esperando
			IF xLe THEN
				eEstado := enum_LeituradosNomes.eAbreConexao;
			END_IF
			
		
		enum_LeituradosNomes.eAbreConexao: //abre conexao
			IF fbSqlDatabase.Connect(INT_TO_UDINT(iNumeroDataBase)) THEN
				IF fbSqlDatabase.bError THEN
					{error <'Não conseguiu abrir a conexao no banco do bloco FB_IniciaOsBlocosDeConfigDoMotor 1'>}
					IF fbSqlDatabase.ipTcResult.ipSourceInfo.sName = 'ADSERR_DEVICE_LICENSENOTFOUND' THEN
						// se der isso ele nao fica tentando e gerando uma caralhada de erro pq nao tem a lisença
						eEstado := enum_LeituradosNomes.eParado;
					ELSE
						eEstado := enum_LeituradosNomes.eAbreConexao;
					END_IF
					
				ELSE
					IF fbSqlDatabase.bConnected THEN
						eEstado := enum_LeituradosNomes.eLeOsNomes;
					END_IF
				END_IF
			END_IF

			
			enum_LeituradosNomes.eLeOsNomes: // le o role
				TagAProcurar		:= sTag1;
				stPara.eParaType	:= E_ExpParameterType.STRING_;
				stPara.nParaSize	:= SIZEOF(TagAProcurar);
				stPara.sParaName	:= 'Tag';
		
				diBaixo	:= LOWER_BOUND(stTelerruptor, 1);
				diCima		:= UPPER_BOUND(stTelerruptor, 1);
		
				// set command with placeholder
				sCmd := CONCAT(CONCAT('SELECT * FROM geral.', sNomeDataBase), ';');
		
				// call functionblock
				IF fbPLCDBCmd.ExecuteDataReturn
					(
						hDBID := INT_TO_UDINT(iNumeroDataBase),
							pExpression := ADR(sCmd),
							cbExpression := SIZEOF(sCmd),
							pData := ADR(TagAProcurar),
							cbData := SIZEOF(TagAProcurar),
							pParameter := ADR(stPara),
							cbParameter := SIZEOF(stPara),
							nStartIndex := DINT_TO_UDINT(diBaixo),
							nRecordCount := DINT_TO_UDINT(diCima),
							pReturnData := ADR(EstruturaBancoLe),
							cbReturnData := SIZEOF(EstruturaBancoLe),
							pRecords := ADR(nRecords))
				THEN
					IF fbPLCDBCmd.bError THEN
						sMensagemErro1 := 'Nao conseguiu a tag';
						{error <'Não conseguiu ler o banco no bloco FB_IniciaOsBlocosDeConfigDoTelerruptor'>}
					ELSE
						sMensagemErro1	:= 'Conseguiu a tag';
						eEstado			:= enum_LeituradosNomes.eFechaConexao;
		
						FOR i := TO_INT(diBaixo+1) TO TO_INT(diCima) DO
							Anterior[i].Config.sNome_Funcao := CONCAT(CONCAT(EstruturaBancoLe[i-1].Tag, ' - '), EstruturaBancoLe[i-1].Funcao);
							stTelerruptor[i].Config.sNome_Funcao := CONCAT(CONCAT(EstruturaBancoLe[i-1].Tag, ' - '), EstruturaBancoLe[i-1].Funcao);
						END_FOR
						
					END_IF
				END_IF
			
			enum_LeituradosNomes.eFechaConexao: // FechaConexao conexao
				IF fbSqlDatabase.Disconnect() THEN
		
					xLe := FALSE;
					xInicia := FALSE;
		
					IF fbSqlDatabase.bError THEN
						{error <'Não conseguiu abrir a conexao no banco do bloco FB_IniciaOsBlocosDeConfigDoMotor 3'>}
						eEstado := enum_LeituradosNomes.eFechaConexao;
					ELSE
						eEstado := enum_LeituradosNomes.eMonitoraTrocaDeNomes;
					END_IF
				END_IF	

			enum_LeituradosNomes.eMonitoraTrocaDeNomes:
				FOR i := TO_INT(diBaixo) TO TO_INT(diCima) DO
					IF (stTelerruptor[i].Config.sNome_Funcao <> Anterior[i].Config.sNome_Funcao) THEN
						Anterior[i].Config.sNome_Funcao := stTelerruptor[i].Config.sNome_Funcao;
						iIndexGrava := i;
						xGrava := TRUE;
					END_IF
				END_FOR					
END_CASE
END_ACTION

END_FUNCTION_BLOCK

// FBs/Controle/Telerruptor/FB_Telerruptor
FUNCTION_BLOCK FB_Telerruptor
VAR_INPUT
	xLigaIHM					: BOOL;
	xLigaBotoeira				: BOOL;
	xLigaInterruptor			: BOOL;
	xFeedBackTellerruptor		: BOOL;
	rTempoTelerruptorAcionado 	: REAL;
END_VAR
VAR_OUTPUT
	xAcionaTelerruptor 			: BOOL;
END_VAR
VAR
	rtLigaTelerruptor 		: Tc2_Standard.R_TRIG;
	rtBotoeira				: Tc2_Standard.R_TRIG;
	rtFotoCelula			: Tc2_Standard.R_TRIG;
	ftDesligaTelerruptor 	: Tc2_Standard.F_TRIG;
	ftFotoCelula			: Tc2_Standard.F_TRIG;
	tonDesligaTelerruptor 	: Tc2_Standard.TON;
END_VAR


IF xLicensaValida87208720 THEN
	
	rtBotoeira(CLK:= xLigaBotoeira, Q=> );
	
	rtLigaTelerruptor(CLK:= xLigaIHM, Q=> );
	ftDesligaTelerruptor(CLK:= xLigaIHM, Q=> );
	
	rtFotoCelula(CLK:= xLigaInterruptor, Q=> );
	ftFotoCelula(CLK:= xLigaInterruptor, Q=> );
	
	
	IF (rtLigaTelerruptor.Q AND NOT xFeedBackTellerruptor) OR (rtBotoeira.Q) OR (rtFotoCelula.Q AND NOT xFeedBackTellerruptor) THEN
		xAcionaTelerruptor := TRUE;
	END_IF
	
	
	
	IF (ftDesligaTelerruptor.Q AND xFeedBackTellerruptor) OR (ftFotoCelula.Q AND xFeedBackTellerruptor) THEN
		xAcionaTelerruptor := TRUE;
	END_IF
	
	
	tonDesligaTelerruptor(IN:= xAcionaTelerruptor, PT:= REAL_TO_TIME(rTempoTelerruptorAcionado*1000), Q=> , ET=> );
	
	IF tonDesligaTelerruptor.Q THEN
		xAcionaTelerruptor := FALSE;
	END_IF
	
ELSE
	ValidaLicensa();
END_IF

END_FUNCTION_BLOCK

// FBs/Controle/FB_Cascata
FUNCTION_BLOCK FB_Cascata
VAR_INPUT
	tCascata : TIME;
	xLiga : BOOL; // botao toggle, enquanto estiver true ele ativa o timmer
END_VAR
VAR_IN_OUT
	xCascata : ARRAY[*] OF BOOL;
END_VAR
VAR_OUTPUT
	iProximoALigar : INT := 1; 
	xLigado : BOOL;
END_VAR
VAR
	i : INT;
	tonGeral : TON;
	diTamanhoArray : DINT;
	diTamanhoMinArray : DINT;
	rtLiga : R_TRIG;
	ftLiga : f_TRIG;
END_VAR

//Criado por Tiago B Cunico para o projeto da area suja de montenegro em 10/2020
IF xLicensaValida87208720 THEN
	
	diTamanhoArray := UPPER_BOUND(xCascata,1);
	diTamanhoMinArray := LOWER_BOUND(xCascata,1);
	
	
	rtLiga(CLK:= xliga, Q=> );
	
	IF rtLiga.q THEN // inicia os acionamentos
		xCascata[diTamanhoMinArray] := TRUE;
	END_IF
	
	ftLiga(CLK:= xliga, Q=> );
	
	IF ftLiga.q THEN // faz como se fosse um reset e para tudo
		iProximoALigar := DINT_TO_INT(diTamanhoMinArray);
		FOR i := DINT_TO_INT(diTamanhoMinArray) TO DINT_TO_INT(diTamanhoArray) DO
			xCascata[i] := FALSE;
		END_FOR
	END_IF
	
	
	
	FOR i := DINT_TO_INT(diTamanhoMinArray) TO DINT_TO_INT(diTamanhoArray) DO
		IF NOT xCascata[i] THEN // quando chegar em um dos bits que estiver false ele passa qual bit é para a iQualLigar e pula fora do for
			iProximoALigar := i;
			EXIT;
		END_IF
	END_FOR
	
	IF tonGeral.q THEN // quando der o tempo ele vai jogar true na variavel e no proximo ciclo ele vai testar a proxima a ligar
		xCascata[iProximoALigar] := TRUE;
	END_IF
	
	tonGeral(IN:= NOT xCascata[iProximoALigar] AND xliga, PT:=tCascata , Q=> , ET=> );
	
	xLigado := xCascata[diTamanhoArray];
		
ELSE
	ValidaLicensa();
END_IF

END_FUNCTION_BLOCK

// FBs/Controle/FB_Cascata1Ligado
FUNCTION_BLOCK FB_Cascata1Ligado
VAR_INPUT
	tCascata : TIME;
	xCicla : BOOL; // caso queira que quando ele chegar no ultimo bool ele reinicie 
	xLiga : BOOL; // botao toggle, enquanto estiver true ele ativa o timmer, se for desligado no meio ele mantem os que ja foram ligado ligado, e se voltar o true ele continua de onde parou.
END_VAR
VAR_IN_OUT
	xArray : ARRAY[*] OF BOOL;
END_VAR
VAR_OUTPUT
	iProximoALigar : INT := 1; 
END_VAR
VAR
	i : INT;
	tonGeral : TON;
	diTamanhoArray : DINT;
	diTamanhoMinArray : DINT;
	rtLiga : R_TRIG;
	ftLiga : f_TRIG;
	ftReinicia : F_TRIG;
	xNaoContinua: BOOL; //para o ciclo caso nao queiram queiram que cicle
END_VAR

IF xLicensaValida87208720 THEN
	
	diTamanhoMinArray := LOWER_BOUND(xArray,1);
	diTamanhoArray := UPPER_BOUND(xArray,1);
	
	
		
	rtLiga(CLK:= xliga, Q=> );
	
	IF rtLiga.q THEN // inicia o ciclo
		xArray[TO_INT(diTamanhoMinArray)] := TRUE;
		xNaoContinua := FALSE;
	END_IF
	
	ftLiga(CLK:= xliga, Q=> );
	
	IF ftLiga.q THEN // faz como se fosse um reset e para tudo
		iProximoALigar := TO_INT(diTamanhoMinArray);
		FOR i := TO_INT(diTamanhoMinArray) TO DINT_TO_INT(diTamanhoArray) DO
			xArray[i] := FALSE;
		END_FOR
		xNaoContinua := FALSE;
	END_IF
	
	
		
	FOR i := TO_INT(diTamanhoMinArray) TO TO_INT(diTamanhoArray) DO
		IF xArray[i] THEN // quando chegar em um dos bits que estiver true ele passa qual bit é para a iQualLigar +1  e pula fora do for
			iProximoALigar := i+1;
			EXIT;
		END_IF
	END_FOR
	
	
	IF iProximoALigar > diTamanhoArray THEN // quando ele chegar no fim ele diz que o prox é o primeiro
		iProximoALigar := TO_INT(diTamanhoMinArray);
	END_IF
	
	
	IF tonGeral.q THEN // quando der o tempo ele vai jogar true na variavel e no proximo ciclo ele vai testar a proxima a ligar		
	
		xArray[iProximoALigar] := TRUE;
	
		IF iProximoALigar = diTamanhoMinArray AND xArray[diTamanhoArray] AND NOT xCicla THEN // para quando ele chega no fim e nao for ciclar desligar o ultimo e parar 
			xArray[iProximoALigar] := FALSE;
			xNaoContinua := TRUE;		
		END_IF
		
		xArray[iProximoALigar-1] := FALSE; // desliga o anterior
		
		
		IF iProximoALigar = diTamanhoMinArray THEN // desliga o ultimo quando inicia
			xArray[diTamanhoArray] := FALSE;
		END_IF
	END_IF
	
	tonGeral(IN:= (NOT xArray[iProximoALigar] AND xliga) AND NOT xNaoContinua, PT:=tCascata , Q=> , ET=> );
ELSE
	ValidaLicensa();
END_IF

END_FUNCTION_BLOCK

// FBs/Controle/FB_ContaRPMporPulso
FUNCTION_BLOCK FB_ContaRPMporPulso

VAR_INPUT
	xSensor : BOOL;
	iQuantidadeDePulsos : INT := 2;
	tAmostra : TIME := T#1S;
	iQuantidadeDeAmostras : INT := 10; // quantas amostras para fazer a media do RPM, max de 1000
	
END_VAR
VAR_OUTPUT
	rContagemReal : REAL;
	rContagemEmRPM : REAL;
END_VAR
VAR
	
rContagemAux : REAL;

rtSinal : R_TRIG;

tonGeraReal : TON;

rAmostraReal : ARRAY[1..1000] OF REAL;

i : INT;

END_VAR

IF xLicensaValida87208720 THEN
	
	rtSinal(CLK:= xSensor, Q=> );
	
	IF rtSinal.q THEN
		rContagemAux := rContagemAux +1;
	END_IF
	
	
	IF tonGeraReal.q THEN
		tonGeraReal.IN := FALSE;
		
		rContagemReal := rContagemAux / iQuantidadeDePulsos;
		
		FOR i := iQuantidadeDeAmostras TO 2 BY -1 DO
			
			rAmostraReal[i] := rAmostraReal[i-1];
			
			IF i < 0 THEN
				EXIT;
			END_IF
		END_FOR
		
		rAmostraReal[1] := rContagemReal;
		
		rContagemEmRPM := 0;
		FOR i := 1 TO iQuantidadeDeAmostras DO 	
			rContagemEmRPM := rContagemEmRPM + rAmostraReal[i];
		END_FOR
		
		
		rContagemEmRPM := rContagemEmRPM/iQuantidadeDeAmostras * 60;
		
		rContagemAux := 0;
	END_IF
	
	
	tonGeraReal(IN:= , PT:= tAmostra, Q=> , ET=> );
	
	
	tonGeraReal.IN := TRUE;
ELSE
	ValidaLicensa();
END_IF

END_FUNCTION_BLOCK

// FBs/Controle/FB_ControleTorreLuminosa
FUNCTION_BLOCK FB_ControleTorreLuminosa
VAR_INPUT
	
	xComeca : BOOL;
	
END_VAR
VAR_IN_OUT
	
	iOrdemCorLiga : ARRAY[*] OF INT; // array de qual corres ligam em qual ordem, 0 -> desligado 1 -> vermelho 2 -> amarelo 3 -> verde 4 -> azul 5 -> buzzer, se quiser que mais de um acione ao mesmo tempo so colocar os dois juntos tipo, verde e amarelo é 24 ou 42
	tTempoDeCadaAcionamento : ARRAY[*] OF TIME; // tempo que vai ser usado para cada item do iOrdemCorLiga
	
END_VAR
VAR_OUTPUT
	
	xVermelho : BOOL;
	xAmarelo : BOOL;
	xAzul : BOOL;
	xVerde : BOOL;
	xBuzzer : BOOL;
	xErro : BOOL;
	
END_VAR
VAR
	
	iTamanhoAcionamentos : INT;
	iTamanhoTempos : INT;
	tonGeral : TON;
	iPosicaoAtual : INT;
	xInicaTimer : BOOL;
	rtInicia : R_TRIG;
	iQuantasCasaMaiorNumero : INT;
	i : INT;
	QuemAciona : ARRAY[1..5] OF BOOL;
	NumQuemAciona : ARRAY[1..5] OF INT;
END_VAR

//Criado por Tiago Bortolini Cunico
IF xLicensaValida87208720 THEN
		
	
	
	iTamanhoAcionamentos := DINT_TO_INT(UPPER_BOUND(iOrdemCorLiga,1));
	iTamanhoTempos := DINT_TO_INT(UPPER_BOUND(tTempoDeCadaAcionamento,1));
	
	
	IF iTamanhoAcionamentos <> iTamanhoTempos THEN
		xErro := TRUE;
	ELSE
		xErro := FALSE;
		
		IF NOT xComeca THEN // força desligado para nao ligar sozinho
			xInicaTimer := FALSE;
			xVermelho := FALSE;
			xAmarelo := FALSE;
			xAzul := FALSE;
			xVerde := FALSE;
			xBuzzer := FALSE;
			
		ELSE
		
			rtInicia(CLK:=xComeca , Q=> );
			
			IF rtInicia.q THEN
				xInicaTimer := TRUE;
				iPosicaoAtual := 1;		
			END_IF
			
			IF tonGeral.q THEN // quando ele chegar no final ele se reseta e passa pro proximo tempo
				xInicaTimer := FALSE;
				
				iPosicaoAtual := iPosicaoAtual+1;// aumenta um e se tiver no max ele reinicia
				IF iPosicaoAtual > iTamanhoAcionamentos THEN
					iPosicaoAtual := 1;
				END_IF
				
				// ve quem tem que acionar
				NumQuemAciona[1] :=  iOrdemCorLiga[iPosicaoAtual]/10000;
				NumQuemAciona[2] :=  iOrdemCorLiga[iPosicaoAtual] MOD 10000 / 1000;
				NumQuemAciona[3] :=  iOrdemCorLiga[iPosicaoAtual] MOD 10000 MOD 1000 / 100;
				NumQuemAciona[4] :=  iOrdemCorLiga[iPosicaoAtual] MOD 10000 MOD 1000 MOD 100 /10;
				NumQuemAciona[5] :=  iOrdemCorLiga[iPosicaoAtual] MOD 10000 MOD 1000 MOD 100 MOD 10;
			END_IF
			
			tonGeral(IN:= xInicaTimer, PT:= tTempoDeCadaAcionamento[iPosicaoAtual], Q=> , ET=> );
			
			xInicaTimer := TRUE;// quando ele reiniciar ali em cima ele se auto reinicia aqui
			
	
			
			// Joga a cor pra fora
			xVermelho := FALSE;
			xAmarelo := FALSE;
			xAzul := FALSE;
			xVerde := FALSE;
			xBuzzer := FALSE;
			
			FOR i:=1 TO 5 DO
				CASE NumQuemAciona[i] OF		
					1:
						xVermelho := TRUE;
					2:
						xAmarelo := TRUE;
					3:
						xVerde := TRUE;
					4:	
						xAzul := TRUE;
					5:
						xBuzzer := TRUE;
				END_CASE
			END_FOR
		
		END_IF
		
		
	END_IF	

ELSE
	ValidaLicensa();
END_IF

END_FUNCTION_BLOCK

// FBs/Controle/FB_ControleTorreLuminosaV2
{attribute 'enable_dynamic_creation'}
FUNCTION_BLOCK FB_ControleTorreLuminosaV2 // Aparece onde eu quero?
VAR_INPUT
	
	xComeca : BOOL; // inicia as luzes
		
	tTempoBeepCurto : TIME := T#500MS; // tempo que ele fara quando for false no array xOrdemLiga
	tTempoBeepLong 	: TIME := T#1000MS; // tempo que ele fara quando for true no array xOrdemLiga
	tTempoEntreBeeps: TIME := T#250MS; //tempo que ele fara entre o true e o false no array xOrdemLiga
	
	iLigaBeepLong 	: INT := 125; // quem liga quando der true no array, 0 -> desligado 1 -> vermelho 2 -> amarelo 3 -> verde 4 -> azul 5 -> buzzer, se quiser que mais de um acione ao mesmo tempo so colocar os dois juntos tipo, verde e amarelo é 24 ou 42
	iLigaBeepCurto	: INT := 125; // quem liga quando for false no array, 0 -> desligado 1 -> vermelho 2 -> amarelo 3 -> verde 4 -> azul 5 -> buzzer, se quiser que mais de um acione ao mesmo tempo so colocar os dois juntos tipo, verde e amarelo é 24 ou 42
	iLigaEntreBeeps	: INT := 1; // quem liga quando for entre tru e false no array,0 -> desligado 1 -> vermelho 2 -> amarelo 3 -> verde 4 -> azul 5 -> buzzer, se quiser que mais de um acione ao mesmo tempo so colocar os dois juntos tipo, verde e amarelo é 24 ou 42
	
END_VAR
VAR_IN_OUT
	xOrdemLiga : ARRAY[*] OF BOOL;
END_VAR
VAR_OUTPUT
	
	xVermelho : BOOL;
	xAmarelo : BOOL;
	xAzul : BOOL;
	xVerde : BOOL;
	xBuzzer : BOOL;
	tContandoAgora	: TIME;
	
	
END_VAR
VAR
	
	iTamanhoAcionamentos : INT;
	iTamanhoXOrdemLiga : INT;
	
	tonGeral : TON;
	iPosicaoAtual : INT;
	xInicaTimer : BOOL;
	rtInicia : R_TRIG;
	iQuantasCasaMaiorNumero : INT;
	i : INT;
	QuemAciona : ARRAY[1..5] OF BOOL;
	NumQuemAciona : ARRAY[1..5] OF INT;
	
	
	iOrdemCorLiga : POINTER TO INT := 0; // array de qual corres ligam em qual ordem, 0 -> desligado 1 -> vermelho 2 -> amarelo 3 -> verde 4 -> azul 5 -> buzzer, se quiser que mais de um acione ao mesmo tempo so colocar os dois juntos tipo, verde e amarelo é 24 ou 42
	tTempoDeCadaAcionamento : POINTER TO TIME := 0; // tempo que vai ser usado para cada item do iOrdemCorLiga
	
END_VAR

// Atualizado por Tiago Bortolini Cunico em 27/04/2021 
IF xLicensaValida87208720 THEN

	iTamanhoAcionamentos := DINT_TO_INT(UPPER_BOUND(xOrdemLiga,1) * 2);
	iTamanhoXOrdemLiga := DINT_TO_INT(UPPER_BOUND(xOrdemLiga,1));
	
	
	IF iOrdemCorLiga = 0 THEN
		//Aloca vetor com o tamanho certo
		iOrdemCorLiga	:= __NEW(INT, iTamanhoAcionamentos);	
		
		//Gera o vetor de controle de quem liga
		FOR i := 1 TO iTamanhoXOrdemLiga DO
			// decide se é beep curto ou longo
			IF xOrdemLiga[i] THEN
				iOrdemCorLiga[i+(i-1)] := iLigaBeepLong;
			ELSE
				iOrdemCorLiga[i+(i-1)] := iLigaBeepCurto;	
			END_IF
		END_FOR
		//completa as lacunas com o entre beeps
		FOR i := 2 TO iTamanhoAcionamentos BY 2 DO
			iOrdemCorLiga[i] := iLigaEntreBeeps;
		END_FOR
	
	END_IF
	
	
	
	
	IF tTempoDeCadaAcionamento = 0 THEN
		//Aloca vetor com o tamanho certo
		tTempoDeCadaAcionamento	:= __NEW(TIME,iTamanhoAcionamentos );	
		
		//Gera o vetor de controle de quanto tempo liga
		 FOR i := 1 TO iTamanhoXOrdemLiga DO
			 // decide se é beep curto ou longo
			IF xOrdemLiga[i] THEN
				tTempoDeCadaAcionamento[i+(i-1)] := tTempoBeepLong;
			ELSE
				tTempoDeCadaAcionamento[i+(i-1)] := tTempoBeepCurto;	
			END_IF
		END_FOR
		//completa as lacunas com o entre beeps
		FOR i := 2 TO iTamanhoAcionamentos BY 2 DO
			tTempoDeCadaAcionamento[i] := tTempoEntreBeeps;
		END_FOR
		//pra dar mais tempo no final e o operador perceber que recomeçou o codig
		tTempoDeCadaAcionamento[iTamanhoAcionamentos] := tTempoBeepLong + tTempoBeepCurto;
	
	END_IF
	
	
	
	// parte igual ao V1
	
	IF NOT xComeca THEN // força desligado para nao ligar sozinho
		xInicaTimer := FALSE;
		xVermelho := FALSE;
		xAmarelo := FALSE;
		xAzul := FALSE;
		xVerde := FALSE;
		xBuzzer := FALSE;
		
	ELSE
	
		rtInicia(CLK:=xComeca , Q=> );
		
		IF rtInicia.q THEN
			xInicaTimer := TRUE;
			iPosicaoAtual := 1;	
			
			// ve quem tem que acionar
			NumQuemAciona[1] :=  iOrdemCorLiga[iPosicaoAtual]/10000;
			NumQuemAciona[2] :=  iOrdemCorLiga[iPosicaoAtual] MOD 10000 / 1000;
			NumQuemAciona[3] :=  iOrdemCorLiga[iPosicaoAtual] MOD 10000 MOD 1000 / 100;
			NumQuemAciona[4] :=  iOrdemCorLiga[iPosicaoAtual] MOD 10000 MOD 1000 MOD 100 /10;
			NumQuemAciona[5] :=  iOrdemCorLiga[iPosicaoAtual] MOD 10000 MOD 1000 MOD 100 MOD 10;	
		END_IF
		
		IF tonGeral.q THEN // quando ele chegar no final ele se reseta e passa pro proximo tempo
			xInicaTimer := FALSE;
			
			iPosicaoAtual := iPosicaoAtual+1;// aumenta um e se tiver no max ele reinicia
			IF iPosicaoAtual > iTamanhoAcionamentos THEN
				iPosicaoAtual := 1;
			END_IF
			
			// ve quem tem que acionar
			NumQuemAciona[1] :=  iOrdemCorLiga[iPosicaoAtual]/10000;
			NumQuemAciona[2] :=  iOrdemCorLiga[iPosicaoAtual] MOD 10000 / 1000;
			NumQuemAciona[3] :=  iOrdemCorLiga[iPosicaoAtual] MOD 10000 MOD 1000 / 100;
			NumQuemAciona[4] :=  iOrdemCorLiga[iPosicaoAtual] MOD 10000 MOD 1000 MOD 100 /10;
			NumQuemAciona[5] :=  iOrdemCorLiga[iPosicaoAtual] MOD 10000 MOD 1000 MOD 100 MOD 10;
		END_IF
		
		tonGeral(IN:= xInicaTimer, PT:= tTempoDeCadaAcionamento[iPosicaoAtual], Q=> , ET=> tContandoAgora);
		xInicaTimer := TRUE;// quando ele reiniciar ali em cima ele se auto reinicia aqui
	
		
		
		// Joga a cor pra fora
		xVermelho := FALSE;
		xAmarelo := FALSE;
		xAzul := FALSE;
		xVerde := FALSE;
		xBuzzer := FALSE;
		
		//ve quem tem que acionar e aciona
		FOR i:=1 TO 5 DO
			CASE NumQuemAciona[i] OF		
				1:
					xVermelho := TRUE;
				2:
					xAmarelo := TRUE;
				3:
					xVerde := TRUE;
				4:	
					xAzul := TRUE;
				5:
					xBuzzer := TRUE;
			END_CASE
		END_FOR
	
	END_IF
	
	
	__DELETE(iOrdemCorLiga);
	iOrdemCorLiga := 0;
	
	__DELETE(tTempoDeCadaAcionamento);
	tTempoDeCadaAcionamento := 0;

ELSE
	ValidaLicensa();
END_IF

END_FUNCTION_BLOCK

// FBs/Controle/FB_TriggerDuplo
FUNCTION_BLOCK FB_TriggerDuplo
VAR_INPUT
	CLK	: BOOL;
END_VAR
VAR_OUTPUT
	Q 	: BOOL;
END_VAR
VAR
	
	rT : R_TRIG;
	fT : F_TRIG;


END_VAR

IF xLicensaValida87208720 THEN
	
	rT(CLK:=CLK);
	fT(CLK:=CLK);
	
	Q := rT.Q OR fT.Q;
	
ELSE
	ValidaLicensa();
END_IF

END_FUNCTION_BLOCK

// FBs/CSV/FB_ControleCSV
FUNCTION_BLOCK FB_ControleCSV
VAR_IN_OUT
	xLeCSV 						: BOOL;
	xEscreveCSV 				: BOOL;
	xEscolhidoArquivo			: BOOL;
	dataBase					: ARRAY[*,*] OF STRING(255);
END_VAR
VAR_INPUT
	sCaminhoBase 				: STRING := 'C:\CSV';
	sCaminhoFinal 				: STRING := '\Sensores Digitais';
	sNomeArquivo				: STRING := '\SensoresDigitais_';
	sArquivosSelecionado		: STRING(255);
	stHoraAgora					: TIMESTRUCT;
END_VAR
VAR_OUTPUT
	xEscritaOcupado 			: BOOL;
	xLeituraOcupado 			: BOOL;
	
	iTotalLeitura 				: INT;
	iAtualLeitura 				: INT;
	iTotalEscrita 				: INT;
	iAtualEscrita 				: INT;
	sArquivos					: ARRAY[1..20]  OF STRING(255);
	
	sStado : eStatusCSV;
END_VAR
VAR
	

	
	fbEscreve : FB_EscreveCSV;
	fbCriaEstruta: FB_CreateDir;
	sNomeAtual : STRING;
	rtComecaEscrever : R_TRIG;
	ftTerminouLer : F_TRIG;
	
	
	fbLeArquivos : FB_EnumFindFileList;
	filesList 	: ARRAY[1..20]  OF ST_FindFileEntry;
	fbLe : FB_LeCSV;
	xLe : BOOL;
	
	sAux : ARRAY[1..20] OF STRING(255);
	sAux2 : ARRAY[1..4] OF STRING(255);
	i : INT;


END_VAR

IF xLicensaValida87208720 THEN

	ExecutaEstado();
	TrocaEstado();

ELSE
	ValidaLicensa();
END_IF

ACTION ExecutaEstado:


CASE sStado OF
	
	Esperando:
	
		fbCriaEstruta(
			sNetId:= ,
			bExecute:= FALSE,  
			bBusy=> , 
			bError=> , 
			nErrId=> );
		

	ChecandoCaminhoGeral:
	
		fbCriaEstruta(
			sNetId:= '', 
			sPathName:= (sCaminhoBase), 
			ePath:= PATH_GENERIC, 
			bExecute:= TRUE, 
			tTimeout:= T#5S, 
			bBusy=> , 
			bError=> , 
			nErrId=> );
			
			
	ChecandoCaminhoEspecifico:
	
		fbCriaEstruta(
			sNetId:= '', 
			sPathName:= CONCAT(sCaminhoBase,sCaminhoFinal), 
			ePath:= PATH_GENERIC, 
			bExecute:= TRUE, 
			tTimeout:= T#5S, 
			bBusy=> , 
			bError=> , 
			nErrId=> );
	
			
	Gravando:
	
		rtComecaEscrever(CLK:= xEscreveCSV, Q=> );

		IF rtComecaEscrever.q THEN

			sAux[1] := CONCAT(sCaminhoFinal,sNomeArquivo);
			sAux[2] := TO_STRING(stHoraAgora.wYear);
			sAux[3] := 'A_';
			sAux[4] := TO_STRING(stHoraAgora.wMonth);
			sAux[5] := 'M_';
			sAux[6] := TO_STRING(stHoraAgora.wDay);
			sAux[7] := 'D_';
			sAux[8] := TO_STRING(stHoraAgora.wHour);
			sAux[9] := 'h_';
			sAux[10] := TO_STRING(stHoraAgora.wMinute);
			sAux[20] := '.csv';
			
			sNomeAtual := concat(sCaminhoBase,F_concatArray(sAux));
		END_IF
			
		
		
		fbEscreve(
			bInicia:= xEscreveCSV, 
			sCaminhoENome:= sNomeAtual, 
			xEscrevePorCima:= TRUE, 
			database:= dataBase, 
			bBusy=> xEscritaOcupado, 
			bError=> , 
			nErrId=> ,
			iTotal=>iTotalEscrita,
			iAgora=>iAtualEscrita);
		
		
		
	lendoArquivos:
	
		IF xLe THEN
			fbLeArquivos.eCmd := eEnumCmd_First;
		ELSE
			fbLeArquivos.eCmd := eEnumCmd_Next;	
		END_IF
		
		
		fbLeArquivos(// e os arquivos da pasta
			sNetId:= '', 
			sPathName:= CONCAT(CONCAT(sCaminhoBase,sCaminhoFinal),'\*.CSV'), 
			eCmd:= , 
			pFindList:= ADR(filesList), 
			cbFindList:= SIZEOF( filesList), 
			bExecute:= xLe, 
			tTimeout:= , 
			bBusy=> , 
			bError=> , 
			nErrID=> , 
			bEOE=> , 
			nFindFiles=> );
		
		xLe := FALSE;
		
		FOR i := 1 TO 20 DO
			sArquivos[i] := filesList[i].sFileName;	
		END_FOR
	

	Lendo:
		// faz a leitura do CSV dos sensores confrme foi escolhido
		
		sAux2[1] := sCaminhoBase;
		sAux2[2] := sCaminhoFinal;
		sAux2[3] := '\';
		sAux2[4] := sArquivosSelecionado;

		fbLe(
			bInicia:= xLeCSV, 
			sCaminhoENome:= F_ConcatArray(sAux2), 
			database:= dataBase, 
			bBusy=> XLeituraOcupado, 
			bError=> , 
			nErrId=> , 
			iTotal=> iTotalLeitura, 
			iAgora=> iAtualLeitura);
		
	
	
	Erro:
		i := i;// so nao dar warning

END_CASE
END_ACTION

ACTION TrocaEstado:



CASE sStado OF
	
	Esperando:
	
		IF xLeCSV OR xEscreveCSV THEN
			xLe := TRUE;
			sStado := ChecandoCaminhoGeral;
		END_IF
	
	ChecandoCaminhoGeral:
	
		IF NOT fbCriaEstruta.bBusy THEN
			sStado := ChecandoCaminhoEspecifico;
			fbCriaEstruta(bExecute:= FALSE);
		END_IF
	
		
		
	ChecandoCaminhoEspecifico:
		// espera terminar o bloco que cria a pasta 
		// ai ele vai ou pra ler sensores ou pra gravar eles
		IF NOT fbCriaEstruta.bBusy THEN
			fbCriaEstruta(bExecute:= FALSE);
			IF xLeCSV THEN
				sStado := lendoArquivos;
			ELSE
				sStado := Gravando;
				rtComecaEscrever(CLK:=FALSE);
				fbEscreve(bInicia:=FALSE);
			END_IF
		END_IF
	
		
	Gravando:
		IF NOT fbEscreve.bBusy THEN
			xEscreveCSV := FALSE;
			sStado := Esperando;
		END_IF
	
	
	lendoArquivos:
	
		IF xEscolhidoArquivo THEN
			sStado := Lendo;
			xEscolhidoArquivo := false;
		END_IF
	

	Lendo:
		// quando terminar de ler ele joga no sensores
		ftTerminouLer(CLK:= fbLe.bBusy, Q=> );
		IF ftTerminouLer.q THEN
			xLeCSV := FALSE;
			sStado := Esperando;
		END_IF
	
	
	
	Erro:
		i := i;// so nao dar warning
	

END_CASE
END_ACTION

END_FUNCTION_BLOCK

// FBs/CSV/FB_EscreveCSV
FUNCTION_BLOCK FB_EscreveCSV
VAR_INPUT
	bInicia : BOOL;
	//sNetId		: T_AmsNetId;	(* TwinCAT system network address *)
	sCaminhoENome	: T_MaxString;(* CSV destination file path and name *)
	xEscrevePorCima : BOOL;
END_VAR
VAR_IN_OUT
	database : ARRAY[*,*] OF STRING(255);
END_VAR
VAR_OUTPUT
	bBusy			: BOOL;
	bError			: BOOL;
	nErrId			: UDINT;
	iTotal			: INT;
	iAgora			: INT;
END_VAR
VAR
	bWrite			: BOOL := FALSE;(* Rising edge starts program execution *)
	sCSVLine		: STRING(1000) := '';(* Single CSV text line (row, record), we are using string as record buffer (your are able to see created fields) *)
	sCSVField		: T_MaxString := '';(* Single CSV field value (column, record field) *)
	nRow	 		: UDINT 	:= 0;(* Row number (record) *)
	nColumn		: UDINT 	:= 0;(* Column number (record field) *)
	hFile			: UINT		:= 0;(* File handle of the source file *)
	step			: DWORD 	:= 0;
	fbFileOpen	: FB_FileOpen;(* Opens file *)
	fbFileClose	: FB_FileClose;(* Closes file *)
	fbFilePuts		: FB_FilePuts;(* Writes one record (line) *)
	fbWriter		: FB_CSVMemBufferWriter;(* Helper function block used to create CSV data bytes (single record line) *)
	rtInicia		: R_TRIG;
	
	MIN_CSV_ROWS : UDINT := 100;
	MIN_CSV_COLUMNS : UDINT := 5;
	MAX_CSV_ROWS : UDINT := 100;
	MAX_CSV_COLUMNS : UDINT := 5;
	MAX_CSV_FIELD_LENGTH : UDINT := 255;
	
	sAux : STRING;
END_VAR

IF xLicensaValida87208720 THEN
//Criado por Tiago Bortolini Cunico
	
	MIN_CSV_ROWS := DINT_TO_UDINT(LOWER_BOUND(database,1));
	MAX_CSV_ROWS := DINT_TO_UDINT(UPPER_BOUND(database,1));
	
	MIN_CSV_COLUMNS :=  DINT_TO_UDINT (LOWER_BOUND(database,2));
	MAX_CSV_COLUMNS := DINT_TO_UDINT (UPPER_BOUND(database,2));
	
	iTotal := TO_INT(MAX_CSV_ROWS);
	
	
	CASE step OF
		0:	(* Wait for rising edge at bWrite variable *)
			rtInicia(CLK:=bInicia , Q=> );//gera borda de subina quando liga	
			IF rtInicia.q THEN
				bWrite := TRUE;
			END_IF
			
			IF bWrite THEN
				bWrite 		:= FALSE;
				bBusy 		:= TRUE;
				bError		:= FALSE;
				nErrId		:= 0;
				hFile		:= 0;
				nRow	 	:= MIN_CSV_ROWS;// se nao ele vai ler lixo
				nColumn		:= MIN_CSV_COLUMNS;
				step 		:= 1;
			END_IF
	
		1:	(* Open source file *)
			fbFileOpen(  bExecute := FALSE  );
			IF xEscrevePorCima THEN
				fbFileOpen( 	sNetId := '', sPathName := sCaminhoENome, nMode := FOPEN_MODEWRITE OR FOPEN_MODETEXT,(* Open file in TEXT mode!   FOPEN_MODEWRITE OR FOPEN_MODETEXT*)
							ePath := PATH_GENERIC, bExecute := TRUE );
			ELSE
				fbFileOpen( 	sNetId := '', sPathName := sCaminhoENome, nMode := FOPEN_MODEAPPEND OR FOPEN_MODETEXT,(* Open file in TEXT mode!   FOPEN_MODEWRITE OR FOPEN_MODETEXT*)
							ePath := PATH_GENERIC, bExecute := TRUE );
			END_IF
			
			step := 2;
	
		2:(* Wait until open not busy *)
			fbFileOpen( bExecute := FALSE, bError => bError, nErrID => nErrID, hFile => hFile );
			IF NOT fbFileOpen.bBusy THEN
				IF NOT fbFileOpen.bError THEN
					step := 3;
				ELSE(* Error: file not found? *)
					step := 100;
				END_IF
			END_IF
	
		3:(* Convert one PLC record to CSV format *)
			sCSVLine := '';
			fbWriter.eCmd := eEnumCmd_First;(* Write first field value *)
			IF nRow <= MAX_CSV_ROWS THEN
	
				FOR nColumn := MIN_CSV_COLUMNS TO MAX_CSV_COLUMNS BY 1 DO
					//IF database[nRow, nColumn] <>  '' THEN //essa linha na real buga o role quando tu tem uma string que tu nao usa no fim do teu database, foda viu
						sCSVField := STRING_TO_CSVFIELD( database[ nRow, nColumn ], FALSE );(* TODO: Get field value from your application *)
		
						(* Add new field to the record buffer *)
						fbWriter( 	pBuffer := ADR( sCSVLine ), cbBuffer := SIZEOF( sCSVLine ) - 1, putValue := sCSVField, pValue := 0, cbValue := 0,
									bCRLF := ( nColumn = MAX_CSV_COLUMNS ) );(* bCRLF == TRUE => Write CRLF after the last field value *)
						IF fbWriter.bOk THEN
							fbWriter.eCmd := eEnumCmd_Next;(* Write next field value *)
						ELSE(* Error *)
							step := 100;
							RETURN;
						END_IF
					//END_IF
				END_FOR(* FOR nColumn := 0... *)
	
				(* FB_FilePuts adds allready CR (carriage return) to the written line.
				We have to replace the $R$L characters with $L character to avoid double CR. *)
				
				IF RIGHT( sCSVLine, 2 ) = '$R$L' THEN
					sCSVLine := REPLACE( sCSVLine, '$L', 2, LEN( sCSVLine ) - 1 );
				END_IF
				
				nRow := nRow + 1;(* Increment number of created records (rows) *)
				iAgora := TO_INT(nRow);
				step := 4;(* Write record to the file *)
	
			ELSE(* All rows written => Close file *)
				step := 10;
			END_IF
	
		4:	(* Write single text line *)
			fbFilePuts( bExecute := FALSE );
			fbFilePuts( sNetId := '', hFile := hFile, sLine := sCSVLine, bExecute := TRUE );
			step := 5;
	
		5:(* Wait until write not busy *)
			fbFilePuts( bExecute := FALSE, bError => bError, nErrID => nErrID );
			IF NOT fbFilePuts.bBusy THEN
				IF NOT fbFilePuts.bError THEN
					step := 3;(* Write next record *)
				ELSE(* Error *)
					step := 100;
				END_IF
			END_IF
	
		10:	(* Close source file *)
			fbFileClose( bExecute := FALSE );
			fbFileClose( sNetId := '', hFile := hFile, bExecute := TRUE );
			step := 11;
	
		11:(* Wait until close not busy *)
			fbFileClose( bExecute := FALSE, bError => bError, nErrID => nErrID );
			IF ( NOT fbFileClose.bBusy ) THEN
				hFile := 0;
				step := 100;
			END_IF
	
		100: (* Error or ready step => cleanup *)
			IF ( hFile <> 0 ) THEN
				step := 10; (* Close the source file *)
			ELSE
				bBusy := FALSE;
				step := 0;	(* Ready *)
			END_IF
	
	END_CASE
ELSE
	ValidaLicensa();
END_IF

END_FUNCTION_BLOCK

// FBs/CSV/FB_LeCSV
FUNCTION_BLOCK FB_LeCSV
VAR_INPUT
	bInicia : BOOL;
	//sNetId		: T_AmsNetId;	(* TwinCAT system network address *)
	sCaminhoENome	: T_MaxString;(* CSV destination file path and name *)
	//xEscrevePorCima : BOOL;
END_VAR
VAR_IN_OUT
	database : ARRAY[*,*] OF STRING(255);
END_VAR
VAR_OUTPUT
	bBusy			: BOOL;
	bError			: BOOL;
	nErrId			: UDINT;
	iTotal			: INT;
	iAgora			: INT;
END_VAR
VAR
	bWrite			: BOOL := FALSE;(* Rising edge starts program execution *)
	sCSVLine		: T_MaxString := '';(* Single CSV text line (row, record), we are using string as record buffer (your are able to see created fields) *)
	sCSVField		: T_MaxString := '';(* Single CSV field value (column, record field) *)
	nRow	 		: UDINT 	:= 0;(* Row number (record) *)
	nColumn		: UDINT 	:= 0;(* Column number (record field) *)
	hFile			: UINT		:= 0;(* File handle of the source file *)
	step			: DWORD 	:= 0;
	fbFileOpen	: FB_FileOpen;(* Opens file *)
	fbFileClose	: FB_FileClose;(* Closes file *)
	fbFilePuts		: FB_FilePuts;(* Writes one record (line) *)
	fbWriter		: FB_CSVMemBufferWriter;(* Helper function block used to create CSV data bytes (single record line) *)
	rtInicia		: R_TRIG;
	
	fbFileGets		: FB_FileGets;(* Reads one record (line) *)
	fbReader		: FB_CSVMemBufferReader;(* Helper function block used to parse CSV data bytes (single record line) *)
	
	MIN_CSV_ROWS : UDINT := 100;
	MIN_CSV_COLUMNS : UDINT := 5;
	MAX_CSV_ROWS : UDINT := 100;
	MAX_CSV_COLUMNS : UDINT := 5;
	MAX_CSV_FIELD_LENGTH : UDINT := 255;
END_VAR

IF xLicensaValida87208720 THEN
		
	
	//Criado por Tiago Bortolini Cunico em 21/10/2021
	
	MIN_CSV_ROWS := DINT_TO_UDINT(LOWER_BOUND(database,1));
	MAX_CSV_ROWS := DINT_TO_UDINT(UPPER_BOUND(database,1));
	
	MIN_CSV_COLUMNS :=  DINT_TO_UDINT (LOWER_BOUND(database,2));
	MAX_CSV_COLUMNS := DINT_TO_UDINT (UPPER_BOUND(database,2));
	
	
	iTotal := TO_INT(MAX_CSV_ROWS);
	
	
	CASE step OF
		0:	(* Wait for rising edge at bRead variable *)
			IF bInicia THEN
				bInicia 	:= FALSE;
				bBusy 		:= TRUE;
				bError		:= FALSE;
				nErrId		:= 0;
				hFile		:= 0;
				nRow	 	:= MIN_CSV_ROWS;
				nColumn		:= MIN_CSV_COLUMNS;
				MEMSET( ADR( database ), 0, SIZEOF( database ) );
				step 		:= 1;
			END_IF
	
		1:	(* Open source file *)
			fbFileOpen(  bExecute := FALSE  );
			fbFileOpen( 	sNetId := '', sPathName := sCaminhoENome, nMode := FOPEN_MODEREAD OR FOPEN_MODETEXT,(* Open file in TEXT mode! *)
							ePath := PATH_GENERIC, bExecute := TRUE );
			step := 2;
	
		2:(* Wait until open not busy *)
			fbFileOpen( bExecute := FALSE, bError => bError, nErrID => nErrID, hFile => hFile );
			IF NOT fbFileOpen.bBusy THEN
				IF NOT fbFileOpen.bError THEN
					step := 3;
				ELSE(* Error: file not found? *)
					step := 100;
				END_IF
			END_IF
	
		3:	(* Read single line (record) *)
			fbFileGets( bExecute := FALSE );
			fbFileGets( sNetId := '', hFile := hFile, bExecute := TRUE );
			step := 4;
	
		4:(* Wait until read not busy *)
			fbFileGets( bExecute := FALSE, bError => bError, nErrID => nErrID, sLine => sCSVLine );
			IF NOT fbFileGets.bBusy THEN
				IF NOT fbFileGets.bError THEN
					IF fbFileGets.bEOF THEN
						step := 10;(* End of file reached => Close source file *)
					ELSE
	
						(* FB_FileGets returns text line without the CR (carriage return) character.
						We have to restore the CR character (replace the $L character with $R$L characters) *)
						IF RIGHT( sCSVLine, 1 ) = '$L' THEN
							sCSVLine := REPLACE( sCSVLine, '$R$L', 2, LEN( sCSVLine ) );
						END_IF
	
						step := 5;
					END_IF
				ELSE(* Error *)
					step := 100;
				END_IF
			END_IF
	
		5:(* Parse single line (record) *)
			fbReader.eCmd := eEnumCmd_First;(* Read first field value *)
			REPEAT
				fbReader( pBuffer := ADR( sCSVLine ), cbBuffer := SIZEOF( sCSVLine ), getValue =>sCSVField );
				IF fbReader.bOk THEN
					fbReader.eCmd := eEnumCmd_Next;(* Read next field value *)
	
					IF ( nRow <= MAX_CSV_ROWS ) THEN
						IF ( nColumn <= MAX_CSV_COLUMNS ) THEN
							database[nRow, nColumn] := CSVFIELD_TO_STRING( sCSVField, FALSE );(* TODO: Save or use the field value in your application *)
						END_IF
					END_IF
	
					nColumn := nColumn + 1;(* Increment number of read columns *)
					IF fbReader.bCRLF THEN(* CRLF == TRUE => End of reacord reached *)
						nRow 		:= nRow + 1;(* Increment number of read records *)
						nColumn 	:= MIN_CSV_COLUMNS;(* Reset number of columns *)
						iAgora 		:= TO_INT(nRow);
					END_IF
	
				ELSE(* Error: End of record reached or all fields read *)
					step := 3;(* Try to read next line *)
				END_IF
			UNTIL NOT fbReader.bOk
			END_REPEAT
	
		10:	(* Close source file *)
			fbFileClose( bExecute := FALSE );
			fbFileClose( sNetId := '', hFile := hFile, bExecute := TRUE );
			step := 11;
	
		11:(* Wait until close not busy *)
			fbFileClose( bExecute := FALSE, bError => bError, nErrID => nErrID );
			IF ( NOT fbFileClose.bBusy ) THEN
				hFile := 0;
				step := 100;
			END_IF
	
